;FOLD SLIN P257 Vel=1 m/s CPDAT257 Tool[4]:Microflown3D Base[0];%{PE}
;FOLD Parameters ;%{h}
;Params IlfProvider=kukaroboter.basistech.inlineforms.movement.spline; Kuka.IsGlobalPoint=False; Kuka.PointName=P257; Kuka.BlendingEnabled=False; Kuka.MoveDataName=CPDAT257; Kuka.VelocityPath=1.000; Kuka.VelocityFieldEnabled=True; Kuka.ColDetectFieldEnabled=True; Kuka.CurrentCDSetIndex=0; Kuka.MovementParameterFieldEnabled=True; IlfCommand=SLIN
;ENDFOLD
SLIN XP257 WITH $VEL = SVEL_CP(2.0, , LCPDAT257),$TOOL = STOOL2(FP257),$BASE = SBASE(FP257.BASE_NO),$IPO_MODE = SIPO_MODE(FP257.IPO_FRAME),$LOAD = SLOAD(FP257.TOOL_NO),$ACC = SACC_CP(LCPDAT257),$ORI_TYPE = SORI_TYP(LCPDAT257),$APO = SAPO(LCPDAT257),$JERK = SJERK(LCPDAT257),$COLLMON_TOL_PRO[1] = USE_CM_PRO_VALUES(0)
;ENDFOLD

;FOLD SLIN P258 Vel=1 m/s CPDAT258 Tool[4]:Microflown3D Base[0];%{PE}
;FOLD Parameters ;%{h}
;Params IlfProvider=kukaroboter.basistech.inlineforms.movement.spline; Kuka.IsGlobalPoint=False; Kuka.PointName=P258; Kuka.BlendingEnabled=False; Kuka.MoveDataName=CPDAT258; Kuka.VelocityPath=1.000; Kuka.VelocityFieldEnabled=True; Kuka.ColDetectFieldEnabled=True; Kuka.CurrentCDSetIndex=0; Kuka.MovementParameterFieldEnabled=True; IlfCommand=SLIN
;ENDFOLD
SLIN XP258 WITH $VEL = SVEL_CP(2.0, , LCPDAT258),$TOOL = STOOL2(FP258),$BASE = SBASE(FP258.BASE_NO),$IPO_MODE = SIPO_MODE(FP258.IPO_FRAME),$LOAD = SLOAD(FP258.TOOL_NO),$ACC = SACC_CP(LCPDAT258),$ORI_TYPE = SORI_TYP(LCPDAT258),$APO = SAPO(LCPDAT258),$JERK = SJERK(LCPDAT258),$COLLMON_TOL_PRO[1] = USE_CM_PRO_VALUES(0)
;ENDFOLD

;FOLD SLIN P259 Vel=1 m/s CPDAT259 Tool[4]:Microflown3D Base[0];%{PE}
;FOLD Parameters ;%{h}
;Params IlfProvider=kukaroboter.basistech.inlineforms.movement.spline; Kuka.IsGlobalPoint=False; Kuka.PointName=P259; Kuka.BlendingEnabled=False; Kuka.MoveDataName=CPDAT259; Kuka.VelocityPath=1.000; Kuka.VelocityFieldEnabled=True; Kuka.ColDetectFieldEnabled=True; Kuka.CurrentCDSetIndex=0; Kuka.MovementParameterFieldEnabled=True; IlfCommand=SLIN
;ENDFOLD
SLIN XP259 WITH $VEL = SVEL_CP(2.0, , LCPDAT259),$TOOL = STOOL2(FP259),$BASE = SBASE(FP259.BASE_NO),$IPO_MODE = SIPO_MODE(FP259.IPO_FRAME),$LOAD = SLOAD(FP259.TOOL_NO),$ACC = SACC_CP(LCPDAT259),$ORI_TYPE = SORI_TYP(LCPDAT259),$APO = SAPO(LCPDAT259),$JERK = SJERK(LCPDAT259),$COLLMON_TOL_PRO[1] = USE_CM_PRO_VALUES(0)
;ENDFOLD

;FOLD SLIN P260 Vel=1 m/s CPDAT260 Tool[4]:Microflown3D Base[0];%{PE}
;FOLD Parameters ;%{h}
;Params IlfProvider=kukaroboter.basistech.inlineforms.movement.spline; Kuka.IsGlobalPoint=False; Kuka.PointName=P260; Kuka.BlendingEnabled=False; Kuka.MoveDataName=CPDAT260; Kuka.VelocityPath=1.000; Kuka.VelocityFieldEnabled=True; Kuka.ColDetectFieldEnabled=True; Kuka.CurrentCDSetIndex=0; Kuka.MovementParameterFieldEnabled=True; IlfCommand=SLIN
;ENDFOLD
SLIN XP260 WITH $VEL = SVEL_CP(2.0, , LCPDAT260),$TOOL = STOOL2(FP260),$BASE = SBASE(FP260.BASE_NO),$IPO_MODE = SIPO_MODE(FP260.IPO_FRAME),$LOAD = SLOAD(FP260.TOOL_NO),$ACC = SACC_CP(LCPDAT260),$ORI_TYPE = SORI_TYP(LCPDAT260),$APO = SAPO(LCPDAT260),$JERK = SJERK(LCPDAT260),$COLLMON_TOL_PRO[1] = USE_CM_PRO_VALUES(0)
;ENDFOLD

;FOLD SLIN P261 Vel=1 m/s CPDAT261 Tool[4]:Microflown3D Base[0];%{PE}
;FOLD Parameters ;%{h}
;Params IlfProvider=kukaroboter.basistech.inlineforms.movement.spline; Kuka.IsGlobalPoint=False; Kuka.PointName=P261; Kuka.BlendingEnabled=False; Kuka.MoveDataName=CPDAT261; Kuka.VelocityPath=1.000; Kuka.VelocityFieldEnabled=True; Kuka.ColDetectFieldEnabled=True; Kuka.CurrentCDSetIndex=0; Kuka.MovementParameterFieldEnabled=True; IlfCommand=SLIN
;ENDFOLD
SLIN XP261 WITH $VEL = SVEL_CP(2.0, , LCPDAT261),$TOOL = STOOL2(FP261),$BASE = SBASE(FP261.BASE_NO),$IPO_MODE = SIPO_MODE(FP261.IPO_FRAME),$LOAD = SLOAD(FP261.TOOL_NO),$ACC = SACC_CP(LCPDAT261),$ORI_TYPE = SORI_TYP(LCPDAT261),$APO = SAPO(LCPDAT261),$JERK = SJERK(LCPDAT261),$COLLMON_TOL_PRO[1] = USE_CM_PRO_VALUES(0)
;ENDFOLD

;FOLD SLIN P262 Vel=1 m/s CPDAT262 Tool[4]:Microflown3D Base[0];%{PE}
;FOLD Parameters ;%{h}
;Params IlfProvider=kukaroboter.basistech.inlineforms.movement.spline; Kuka.IsGlobalPoint=False; Kuka.PointName=P262; Kuka.BlendingEnabled=False; Kuka.MoveDataName=CPDAT262; Kuka.VelocityPath=1.000; Kuka.VelocityFieldEnabled=True; Kuka.ColDetectFieldEnabled=True; Kuka.CurrentCDSetIndex=0; Kuka.MovementParameterFieldEnabled=True; IlfCommand=SLIN
;ENDFOLD
SLIN XP262 WITH $VEL = SVEL_CP(2.0, , LCPDAT262),$TOOL = STOOL2(FP262),$BASE = SBASE(FP262.BASE_NO),$IPO_MODE = SIPO_MODE(FP262.IPO_FRAME),$LOAD = SLOAD(FP262.TOOL_NO),$ACC = SACC_CP(LCPDAT262),$ORI_TYPE = SORI_TYP(LCPDAT262),$APO = SAPO(LCPDAT262),$JERK = SJERK(LCPDAT262),$COLLMON_TOL_PRO[1] = USE_CM_PRO_VALUES(0)
;ENDFOLD

;FOLD SLIN P263 Vel=1 m/s CPDAT263 Tool[4]:Microflown3D Base[0];%{PE}
;FOLD Parameters ;%{h}
;Params IlfProvider=kukaroboter.basistech.inlineforms.movement.spline; Kuka.IsGlobalPoint=False; Kuka.PointName=P263; Kuka.BlendingEnabled=False; Kuka.MoveDataName=CPDAT263; Kuka.VelocityPath=1.000; Kuka.VelocityFieldEnabled=True; Kuka.ColDetectFieldEnabled=True; Kuka.CurrentCDSetIndex=0; Kuka.MovementParameterFieldEnabled=True; IlfCommand=SLIN
;ENDFOLD
SLIN XP263 WITH $VEL = SVEL_CP(2.0, , LCPDAT263),$TOOL = STOOL2(FP263),$BASE = SBASE(FP263.BASE_NO),$IPO_MODE = SIPO_MODE(FP263.IPO_FRAME),$LOAD = SLOAD(FP263.TOOL_NO),$ACC = SACC_CP(LCPDAT263),$ORI_TYPE = SORI_TYP(LCPDAT263),$APO = SAPO(LCPDAT263),$JERK = SJERK(LCPDAT263),$COLLMON_TOL_PRO[1] = USE_CM_PRO_VALUES(0)
;ENDFOLD

;FOLD SLIN P264 Vel=1 m/s CPDAT264 Tool[4]:Microflown3D Base[0];%{PE}
;FOLD Parameters ;%{h}
;Params IlfProvider=kukaroboter.basistech.inlineforms.movement.spline; Kuka.IsGlobalPoint=False; Kuka.PointName=P264; Kuka.BlendingEnabled=False; Kuka.MoveDataName=CPDAT264; Kuka.VelocityPath=1.000; Kuka.VelocityFieldEnabled=True; Kuka.ColDetectFieldEnabled=True; Kuka.CurrentCDSetIndex=0; Kuka.MovementParameterFieldEnabled=True; IlfCommand=SLIN
;ENDFOLD
SLIN XP264 WITH $VEL = SVEL_CP(2.0, , LCPDAT264),$TOOL = STOOL2(FP264),$BASE = SBASE(FP264.BASE_NO),$IPO_MODE = SIPO_MODE(FP264.IPO_FRAME),$LOAD = SLOAD(FP264.TOOL_NO),$ACC = SACC_CP(LCPDAT264),$ORI_TYPE = SORI_TYP(LCPDAT264),$APO = SAPO(LCPDAT264),$JERK = SJERK(LCPDAT264),$COLLMON_TOL_PRO[1] = USE_CM_PRO_VALUES(0)
;ENDFOLD

;FOLD SLIN P265 Vel=1 m/s CPDAT265 Tool[4]:Microflown3D Base[0];%{PE}
;FOLD Parameters ;%{h}
;Params IlfProvider=kukaroboter.basistech.inlineforms.movement.spline; Kuka.IsGlobalPoint=False; Kuka.PointName=P265; Kuka.BlendingEnabled=False; Kuka.MoveDataName=CPDAT265; Kuka.VelocityPath=1.000; Kuka.VelocityFieldEnabled=True; Kuka.ColDetectFieldEnabled=True; Kuka.CurrentCDSetIndex=0; Kuka.MovementParameterFieldEnabled=True; IlfCommand=SLIN
;ENDFOLD
SLIN XP265 WITH $VEL = SVEL_CP(2.0, , LCPDAT265),$TOOL = STOOL2(FP265),$BASE = SBASE(FP265.BASE_NO),$IPO_MODE = SIPO_MODE(FP265.IPO_FRAME),$LOAD = SLOAD(FP265.TOOL_NO),$ACC = SACC_CP(LCPDAT265),$ORI_TYPE = SORI_TYP(LCPDAT265),$APO = SAPO(LCPDAT265),$JERK = SJERK(LCPDAT265),$COLLMON_TOL_PRO[1] = USE_CM_PRO_VALUES(0)
;ENDFOLD

;FOLD SLIN P266 Vel=1 m/s CPDAT266 Tool[4]:Microflown3D Base[0];%{PE}
;FOLD Parameters ;%{h}
;Params IlfProvider=kukaroboter.basistech.inlineforms.movement.spline; Kuka.IsGlobalPoint=False; Kuka.PointName=P266; Kuka.BlendingEnabled=False; Kuka.MoveDataName=CPDAT266; Kuka.VelocityPath=1.000; Kuka.VelocityFieldEnabled=True; Kuka.ColDetectFieldEnabled=True; Kuka.CurrentCDSetIndex=0; Kuka.MovementParameterFieldEnabled=True; IlfCommand=SLIN
;ENDFOLD
SLIN XP266 WITH $VEL = SVEL_CP(2.0, , LCPDAT266),$TOOL = STOOL2(FP266),$BASE = SBASE(FP266.BASE_NO),$IPO_MODE = SIPO_MODE(FP266.IPO_FRAME),$LOAD = SLOAD(FP266.TOOL_NO),$ACC = SACC_CP(LCPDAT266),$ORI_TYPE = SORI_TYP(LCPDAT266),$APO = SAPO(LCPDAT266),$JERK = SJERK(LCPDAT266),$COLLMON_TOL_PRO[1] = USE_CM_PRO_VALUES(0)
;ENDFOLD

;FOLD SLIN P267 Vel=1 m/s CPDAT267 Tool[4]:Microflown3D Base[0];%{PE}
;FOLD Parameters ;%{h}
;Params IlfProvider=kukaroboter.basistech.inlineforms.movement.spline; Kuka.IsGlobalPoint=False; Kuka.PointName=P267; Kuka.BlendingEnabled=False; Kuka.MoveDataName=CPDAT267; Kuka.VelocityPath=1.000; Kuka.VelocityFieldEnabled=True; Kuka.ColDetectFieldEnabled=True; Kuka.CurrentCDSetIndex=0; Kuka.MovementParameterFieldEnabled=True; IlfCommand=SLIN
;ENDFOLD
SLIN XP267 WITH $VEL = SVEL_CP(2.0, , LCPDAT267),$TOOL = STOOL2(FP267),$BASE = SBASE(FP267.BASE_NO),$IPO_MODE = SIPO_MODE(FP267.IPO_FRAME),$LOAD = SLOAD(FP267.TOOL_NO),$ACC = SACC_CP(LCPDAT267),$ORI_TYPE = SORI_TYP(LCPDAT267),$APO = SAPO(LCPDAT267),$JERK = SJERK(LCPDAT267),$COLLMON_TOL_PRO[1] = USE_CM_PRO_VALUES(0)
;ENDFOLD

;FOLD SLIN P268 Vel=1 m/s CPDAT268 Tool[4]:Microflown3D Base[0];%{PE}
;FOLD Parameters ;%{h}
;Params IlfProvider=kukaroboter.basistech.inlineforms.movement.spline; Kuka.IsGlobalPoint=False; Kuka.PointName=P268; Kuka.BlendingEnabled=False; Kuka.MoveDataName=CPDAT268; Kuka.VelocityPath=1.000; Kuka.VelocityFieldEnabled=True; Kuka.ColDetectFieldEnabled=True; Kuka.CurrentCDSetIndex=0; Kuka.MovementParameterFieldEnabled=True; IlfCommand=SLIN
;ENDFOLD
SLIN XP268 WITH $VEL = SVEL_CP(2.0, , LCPDAT268),$TOOL = STOOL2(FP268),$BASE = SBASE(FP268.BASE_NO),$IPO_MODE = SIPO_MODE(FP268.IPO_FRAME),$LOAD = SLOAD(FP268.TOOL_NO),$ACC = SACC_CP(LCPDAT268),$ORI_TYPE = SORI_TYP(LCPDAT268),$APO = SAPO(LCPDAT268),$JERK = SJERK(LCPDAT268),$COLLMON_TOL_PRO[1] = USE_CM_PRO_VALUES(0)
;ENDFOLD

;FOLD SLIN P269 Vel=1 m/s CPDAT269 Tool[4]:Microflown3D Base[0];%{PE}
;FOLD Parameters ;%{h}
;Params IlfProvider=kukaroboter.basistech.inlineforms.movement.spline; Kuka.IsGlobalPoint=False; Kuka.PointName=P269; Kuka.BlendingEnabled=False; Kuka.MoveDataName=CPDAT269; Kuka.VelocityPath=1.000; Kuka.VelocityFieldEnabled=True; Kuka.ColDetectFieldEnabled=True; Kuka.CurrentCDSetIndex=0; Kuka.MovementParameterFieldEnabled=True; IlfCommand=SLIN
;ENDFOLD
SLIN XP269 WITH $VEL = SVEL_CP(2.0, , LCPDAT269),$TOOL = STOOL2(FP269),$BASE = SBASE(FP269.BASE_NO),$IPO_MODE = SIPO_MODE(FP269.IPO_FRAME),$LOAD = SLOAD(FP269.TOOL_NO),$ACC = SACC_CP(LCPDAT269),$ORI_TYPE = SORI_TYP(LCPDAT269),$APO = SAPO(LCPDAT269),$JERK = SJERK(LCPDAT269),$COLLMON_TOL_PRO[1] = USE_CM_PRO_VALUES(0)
;ENDFOLD

;FOLD SLIN P270 Vel=1 m/s CPDAT270 Tool[4]:Microflown3D Base[0];%{PE}
;FOLD Parameters ;%{h}
;Params IlfProvider=kukaroboter.basistech.inlineforms.movement.spline; Kuka.IsGlobalPoint=False; Kuka.PointName=P270; Kuka.BlendingEnabled=False; Kuka.MoveDataName=CPDAT270; Kuka.VelocityPath=1.000; Kuka.VelocityFieldEnabled=True; Kuka.ColDetectFieldEnabled=True; Kuka.CurrentCDSetIndex=0; Kuka.MovementParameterFieldEnabled=True; IlfCommand=SLIN
;ENDFOLD
SLIN XP270 WITH $VEL = SVEL_CP(2.0, , LCPDAT270),$TOOL = STOOL2(FP270),$BASE = SBASE(FP270.BASE_NO),$IPO_MODE = SIPO_MODE(FP270.IPO_FRAME),$LOAD = SLOAD(FP270.TOOL_NO),$ACC = SACC_CP(LCPDAT270),$ORI_TYPE = SORI_TYP(LCPDAT270),$APO = SAPO(LCPDAT270),$JERK = SJERK(LCPDAT270),$COLLMON_TOL_PRO[1] = USE_CM_PRO_VALUES(0)
;ENDFOLD

;FOLD SLIN P271 Vel=1 m/s CPDAT271 Tool[4]:Microflown3D Base[0];%{PE}
;FOLD Parameters ;%{h}
;Params IlfProvider=kukaroboter.basistech.inlineforms.movement.spline; Kuka.IsGlobalPoint=False; Kuka.PointName=P271; Kuka.BlendingEnabled=False; Kuka.MoveDataName=CPDAT271; Kuka.VelocityPath=1.000; Kuka.VelocityFieldEnabled=True; Kuka.ColDetectFieldEnabled=True; Kuka.CurrentCDSetIndex=0; Kuka.MovementParameterFieldEnabled=True; IlfCommand=SLIN
;ENDFOLD
SLIN XP271 WITH $VEL = SVEL_CP(2.0, , LCPDAT271),$TOOL = STOOL2(FP271),$BASE = SBASE(FP271.BASE_NO),$IPO_MODE = SIPO_MODE(FP271.IPO_FRAME),$LOAD = SLOAD(FP271.TOOL_NO),$ACC = SACC_CP(LCPDAT271),$ORI_TYPE = SORI_TYP(LCPDAT271),$APO = SAPO(LCPDAT271),$JERK = SJERK(LCPDAT271),$COLLMON_TOL_PRO[1] = USE_CM_PRO_VALUES(0)
;ENDFOLD

;FOLD SLIN P272 Vel=1 m/s CPDAT272 Tool[4]:Microflown3D Base[0];%{PE}
;FOLD Parameters ;%{h}
;Params IlfProvider=kukaroboter.basistech.inlineforms.movement.spline; Kuka.IsGlobalPoint=False; Kuka.PointName=P272; Kuka.BlendingEnabled=False; Kuka.MoveDataName=CPDAT272; Kuka.VelocityPath=1.000; Kuka.VelocityFieldEnabled=True; Kuka.ColDetectFieldEnabled=True; Kuka.CurrentCDSetIndex=0; Kuka.MovementParameterFieldEnabled=True; IlfCommand=SLIN
;ENDFOLD
SLIN XP272 WITH $VEL = SVEL_CP(2.0, , LCPDAT272),$TOOL = STOOL2(FP272),$BASE = SBASE(FP272.BASE_NO),$IPO_MODE = SIPO_MODE(FP272.IPO_FRAME),$LOAD = SLOAD(FP272.TOOL_NO),$ACC = SACC_CP(LCPDAT272),$ORI_TYPE = SORI_TYP(LCPDAT272),$APO = SAPO(LCPDAT272),$JERK = SJERK(LCPDAT272),$COLLMON_TOL_PRO[1] = USE_CM_PRO_VALUES(0)
;ENDFOLD

;FOLD SLIN P273 Vel=1 m/s CPDAT273 Tool[4]:Microflown3D Base[0];%{PE}
;FOLD Parameters ;%{h}
;Params IlfProvider=kukaroboter.basistech.inlineforms.movement.spline; Kuka.IsGlobalPoint=False; Kuka.PointName=P273; Kuka.BlendingEnabled=False; Kuka.MoveDataName=CPDAT273; Kuka.VelocityPath=1.000; Kuka.VelocityFieldEnabled=True; Kuka.ColDetectFieldEnabled=True; Kuka.CurrentCDSetIndex=0; Kuka.MovementParameterFieldEnabled=True; IlfCommand=SLIN
;ENDFOLD
SLIN XP273 WITH $VEL = SVEL_CP(2.0, , LCPDAT273),$TOOL = STOOL2(FP273),$BASE = SBASE(FP273.BASE_NO),$IPO_MODE = SIPO_MODE(FP273.IPO_FRAME),$LOAD = SLOAD(FP273.TOOL_NO),$ACC = SACC_CP(LCPDAT273),$ORI_TYPE = SORI_TYP(LCPDAT273),$APO = SAPO(LCPDAT273),$JERK = SJERK(LCPDAT273),$COLLMON_TOL_PRO[1] = USE_CM_PRO_VALUES(0)
;ENDFOLD

;FOLD SLIN P274 Vel=1 m/s CPDAT274 Tool[4]:Microflown3D Base[0];%{PE}
;FOLD Parameters ;%{h}
;Params IlfProvider=kukaroboter.basistech.inlineforms.movement.spline; Kuka.IsGlobalPoint=False; Kuka.PointName=P274; Kuka.BlendingEnabled=False; Kuka.MoveDataName=CPDAT274; Kuka.VelocityPath=1.000; Kuka.VelocityFieldEnabled=True; Kuka.ColDetectFieldEnabled=True; Kuka.CurrentCDSetIndex=0; Kuka.MovementParameterFieldEnabled=True; IlfCommand=SLIN
;ENDFOLD
SLIN XP274 WITH $VEL = SVEL_CP(2.0, , LCPDAT274),$TOOL = STOOL2(FP274),$BASE = SBASE(FP274.BASE_NO),$IPO_MODE = SIPO_MODE(FP274.IPO_FRAME),$LOAD = SLOAD(FP274.TOOL_NO),$ACC = SACC_CP(LCPDAT274),$ORI_TYPE = SORI_TYP(LCPDAT274),$APO = SAPO(LCPDAT274),$JERK = SJERK(LCPDAT274),$COLLMON_TOL_PRO[1] = USE_CM_PRO_VALUES(0)
;ENDFOLD

;FOLD SLIN P275 Vel=1 m/s CPDAT275 Tool[4]:Microflown3D Base[0];%{PE}
;FOLD Parameters ;%{h}
;Params IlfProvider=kukaroboter.basistech.inlineforms.movement.spline; Kuka.IsGlobalPoint=False; Kuka.PointName=P275; Kuka.BlendingEnabled=False; Kuka.MoveDataName=CPDAT275; Kuka.VelocityPath=1.000; Kuka.VelocityFieldEnabled=True; Kuka.ColDetectFieldEnabled=True; Kuka.CurrentCDSetIndex=0; Kuka.MovementParameterFieldEnabled=True; IlfCommand=SLIN
;ENDFOLD
SLIN XP275 WITH $VEL = SVEL_CP(2.0, , LCPDAT275),$TOOL = STOOL2(FP275),$BASE = SBASE(FP275.BASE_NO),$IPO_MODE = SIPO_MODE(FP275.IPO_FRAME),$LOAD = SLOAD(FP275.TOOL_NO),$ACC = SACC_CP(LCPDAT275),$ORI_TYPE = SORI_TYP(LCPDAT275),$APO = SAPO(LCPDAT275),$JERK = SJERK(LCPDAT275),$COLLMON_TOL_PRO[1] = USE_CM_PRO_VALUES(0)
;ENDFOLD

;FOLD SLIN P276 Vel=1 m/s CPDAT276 Tool[4]:Microflown3D Base[0];%{PE}
;FOLD Parameters ;%{h}
;Params IlfProvider=kukaroboter.basistech.inlineforms.movement.spline; Kuka.IsGlobalPoint=False; Kuka.PointName=P276; Kuka.BlendingEnabled=False; Kuka.MoveDataName=CPDAT276; Kuka.VelocityPath=1.000; Kuka.VelocityFieldEnabled=True; Kuka.ColDetectFieldEnabled=True; Kuka.CurrentCDSetIndex=0; Kuka.MovementParameterFieldEnabled=True; IlfCommand=SLIN
;ENDFOLD
SLIN XP276 WITH $VEL = SVEL_CP(2.0, , LCPDAT276),$TOOL = STOOL2(FP276),$BASE = SBASE(FP276.BASE_NO),$IPO_MODE = SIPO_MODE(FP276.IPO_FRAME),$LOAD = SLOAD(FP276.TOOL_NO),$ACC = SACC_CP(LCPDAT276),$ORI_TYPE = SORI_TYP(LCPDAT276),$APO = SAPO(LCPDAT276),$JERK = SJERK(LCPDAT276),$COLLMON_TOL_PRO[1] = USE_CM_PRO_VALUES(0)
;ENDFOLD

;FOLD SLIN P277 Vel=1 m/s CPDAT277 Tool[4]:Microflown3D Base[0];%{PE}
;FOLD Parameters ;%{h}
;Params IlfProvider=kukaroboter.basistech.inlineforms.movement.spline; Kuka.IsGlobalPoint=False; Kuka.PointName=P277; Kuka.BlendingEnabled=False; Kuka.MoveDataName=CPDAT277; Kuka.VelocityPath=1.000; Kuka.VelocityFieldEnabled=True; Kuka.ColDetectFieldEnabled=True; Kuka.CurrentCDSetIndex=0; Kuka.MovementParameterFieldEnabled=True; IlfCommand=SLIN
;ENDFOLD
SLIN XP277 WITH $VEL = SVEL_CP(2.0, , LCPDAT277),$TOOL = STOOL2(FP277),$BASE = SBASE(FP277.BASE_NO),$IPO_MODE = SIPO_MODE(FP277.IPO_FRAME),$LOAD = SLOAD(FP277.TOOL_NO),$ACC = SACC_CP(LCPDAT277),$ORI_TYPE = SORI_TYP(LCPDAT277),$APO = SAPO(LCPDAT277),$JERK = SJERK(LCPDAT277),$COLLMON_TOL_PRO[1] = USE_CM_PRO_VALUES(0)
;ENDFOLD

;FOLD SLIN P278 Vel=1 m/s CPDAT278 Tool[4]:Microflown3D Base[0];%{PE}
;FOLD Parameters ;%{h}
;Params IlfProvider=kukaroboter.basistech.inlineforms.movement.spline; Kuka.IsGlobalPoint=False; Kuka.PointName=P278; Kuka.BlendingEnabled=False; Kuka.MoveDataName=CPDAT278; Kuka.VelocityPath=1.000; Kuka.VelocityFieldEnabled=True; Kuka.ColDetectFieldEnabled=True; Kuka.CurrentCDSetIndex=0; Kuka.MovementParameterFieldEnabled=True; IlfCommand=SLIN
;ENDFOLD
SLIN XP278 WITH $VEL = SVEL_CP(2.0, , LCPDAT278),$TOOL = STOOL2(FP278),$BASE = SBASE(FP278.BASE_NO),$IPO_MODE = SIPO_MODE(FP278.IPO_FRAME),$LOAD = SLOAD(FP278.TOOL_NO),$ACC = SACC_CP(LCPDAT278),$ORI_TYPE = SORI_TYP(LCPDAT278),$APO = SAPO(LCPDAT278),$JERK = SJERK(LCPDAT278),$COLLMON_TOL_PRO[1] = USE_CM_PRO_VALUES(0)
;ENDFOLD

;FOLD SLIN P279 Vel=1 m/s CPDAT279 Tool[4]:Microflown3D Base[0];%{PE}
;FOLD Parameters ;%{h}
;Params IlfProvider=kukaroboter.basistech.inlineforms.movement.spline; Kuka.IsGlobalPoint=False; Kuka.PointName=P279; Kuka.BlendingEnabled=False; Kuka.MoveDataName=CPDAT279; Kuka.VelocityPath=1.000; Kuka.VelocityFieldEnabled=True; Kuka.ColDetectFieldEnabled=True; Kuka.CurrentCDSetIndex=0; Kuka.MovementParameterFieldEnabled=True; IlfCommand=SLIN
;ENDFOLD
SLIN XP279 WITH $VEL = SVEL_CP(2.0, , LCPDAT279),$TOOL = STOOL2(FP279),$BASE = SBASE(FP279.BASE_NO),$IPO_MODE = SIPO_MODE(FP279.IPO_FRAME),$LOAD = SLOAD(FP279.TOOL_NO),$ACC = SACC_CP(LCPDAT279),$ORI_TYPE = SORI_TYP(LCPDAT279),$APO = SAPO(LCPDAT279),$JERK = SJERK(LCPDAT279),$COLLMON_TOL_PRO[1] = USE_CM_PRO_VALUES(0)
;ENDFOLD

;FOLD SLIN P280 Vel=1 m/s CPDAT280 Tool[4]:Microflown3D Base[0];%{PE}
;FOLD Parameters ;%{h}
;Params IlfProvider=kukaroboter.basistech.inlineforms.movement.spline; Kuka.IsGlobalPoint=False; Kuka.PointName=P280; Kuka.BlendingEnabled=False; Kuka.MoveDataName=CPDAT280; Kuka.VelocityPath=1.000; Kuka.VelocityFieldEnabled=True; Kuka.ColDetectFieldEnabled=True; Kuka.CurrentCDSetIndex=0; Kuka.MovementParameterFieldEnabled=True; IlfCommand=SLIN
;ENDFOLD
SLIN XP280 WITH $VEL = SVEL_CP(2.0, , LCPDAT280),$TOOL = STOOL2(FP280),$BASE = SBASE(FP280.BASE_NO),$IPO_MODE = SIPO_MODE(FP280.IPO_FRAME),$LOAD = SLOAD(FP280.TOOL_NO),$ACC = SACC_CP(LCPDAT280),$ORI_TYPE = SORI_TYP(LCPDAT280),$APO = SAPO(LCPDAT280),$JERK = SJERK(LCPDAT280),$COLLMON_TOL_PRO[1] = USE_CM_PRO_VALUES(0)
;ENDFOLD

;FOLD SLIN P281 Vel=1 m/s CPDAT281 Tool[4]:Microflown3D Base[0];%{PE}
;FOLD Parameters ;%{h}
;Params IlfProvider=kukaroboter.basistech.inlineforms.movement.spline; Kuka.IsGlobalPoint=False; Kuka.PointName=P281; Kuka.BlendingEnabled=False; Kuka.MoveDataName=CPDAT281; Kuka.VelocityPath=1.000; Kuka.VelocityFieldEnabled=True; Kuka.ColDetectFieldEnabled=True; Kuka.CurrentCDSetIndex=0; Kuka.MovementParameterFieldEnabled=True; IlfCommand=SLIN
;ENDFOLD
SLIN XP281 WITH $VEL = SVEL_CP(2.0, , LCPDAT281),$TOOL = STOOL2(FP281),$BASE = SBASE(FP281.BASE_NO),$IPO_MODE = SIPO_MODE(FP281.IPO_FRAME),$LOAD = SLOAD(FP281.TOOL_NO),$ACC = SACC_CP(LCPDAT281),$ORI_TYPE = SORI_TYP(LCPDAT281),$APO = SAPO(LCPDAT281),$JERK = SJERK(LCPDAT281),$COLLMON_TOL_PRO[1] = USE_CM_PRO_VALUES(0)
;ENDFOLD

;FOLD SLIN P282 Vel=1 m/s CPDAT282 Tool[4]:Microflown3D Base[0];%{PE}
;FOLD Parameters ;%{h}
;Params IlfProvider=kukaroboter.basistech.inlineforms.movement.spline; Kuka.IsGlobalPoint=False; Kuka.PointName=P282; Kuka.BlendingEnabled=False; Kuka.MoveDataName=CPDAT282; Kuka.VelocityPath=1.000; Kuka.VelocityFieldEnabled=True; Kuka.ColDetectFieldEnabled=True; Kuka.CurrentCDSetIndex=0; Kuka.MovementParameterFieldEnabled=True; IlfCommand=SLIN
;ENDFOLD
SLIN XP282 WITH $VEL = SVEL_CP(2.0, , LCPDAT282),$TOOL = STOOL2(FP282),$BASE = SBASE(FP282.BASE_NO),$IPO_MODE = SIPO_MODE(FP282.IPO_FRAME),$LOAD = SLOAD(FP282.TOOL_NO),$ACC = SACC_CP(LCPDAT282),$ORI_TYPE = SORI_TYP(LCPDAT282),$APO = SAPO(LCPDAT282),$JERK = SJERK(LCPDAT282),$COLLMON_TOL_PRO[1] = USE_CM_PRO_VALUES(0)
;ENDFOLD

;FOLD SLIN P283 Vel=1 m/s CPDAT283 Tool[4]:Microflown3D Base[0];%{PE}
;FOLD Parameters ;%{h}
;Params IlfProvider=kukaroboter.basistech.inlineforms.movement.spline; Kuka.IsGlobalPoint=False; Kuka.PointName=P283; Kuka.BlendingEnabled=False; Kuka.MoveDataName=CPDAT283; Kuka.VelocityPath=1.000; Kuka.VelocityFieldEnabled=True; Kuka.ColDetectFieldEnabled=True; Kuka.CurrentCDSetIndex=0; Kuka.MovementParameterFieldEnabled=True; IlfCommand=SLIN
;ENDFOLD
SLIN XP283 WITH $VEL = SVEL_CP(2.0, , LCPDAT283),$TOOL = STOOL2(FP283),$BASE = SBASE(FP283.BASE_NO),$IPO_MODE = SIPO_MODE(FP283.IPO_FRAME),$LOAD = SLOAD(FP283.TOOL_NO),$ACC = SACC_CP(LCPDAT283),$ORI_TYPE = SORI_TYP(LCPDAT283),$APO = SAPO(LCPDAT283),$JERK = SJERK(LCPDAT283),$COLLMON_TOL_PRO[1] = USE_CM_PRO_VALUES(0)
;ENDFOLD

;FOLD SLIN P284 Vel=1 m/s CPDAT284 Tool[4]:Microflown3D Base[0];%{PE}
;FOLD Parameters ;%{h}
;Params IlfProvider=kukaroboter.basistech.inlineforms.movement.spline; Kuka.IsGlobalPoint=False; Kuka.PointName=P284; Kuka.BlendingEnabled=False; Kuka.MoveDataName=CPDAT284; Kuka.VelocityPath=1.000; Kuka.VelocityFieldEnabled=True; Kuka.ColDetectFieldEnabled=True; Kuka.CurrentCDSetIndex=0; Kuka.MovementParameterFieldEnabled=True; IlfCommand=SLIN
;ENDFOLD
SLIN XP284 WITH $VEL = SVEL_CP(2.0, , LCPDAT284),$TOOL = STOOL2(FP284),$BASE = SBASE(FP284.BASE_NO),$IPO_MODE = SIPO_MODE(FP284.IPO_FRAME),$LOAD = SLOAD(FP284.TOOL_NO),$ACC = SACC_CP(LCPDAT284),$ORI_TYPE = SORI_TYP(LCPDAT284),$APO = SAPO(LCPDAT284),$JERK = SJERK(LCPDAT284),$COLLMON_TOL_PRO[1] = USE_CM_PRO_VALUES(0)
;ENDFOLD

;FOLD SLIN P285 Vel=1 m/s CPDAT285 Tool[4]:Microflown3D Base[0];%{PE}
;FOLD Parameters ;%{h}
;Params IlfProvider=kukaroboter.basistech.inlineforms.movement.spline; Kuka.IsGlobalPoint=False; Kuka.PointName=P285; Kuka.BlendingEnabled=False; Kuka.MoveDataName=CPDAT285; Kuka.VelocityPath=1.000; Kuka.VelocityFieldEnabled=True; Kuka.ColDetectFieldEnabled=True; Kuka.CurrentCDSetIndex=0; Kuka.MovementParameterFieldEnabled=True; IlfCommand=SLIN
;ENDFOLD
SLIN XP285 WITH $VEL = SVEL_CP(2.0, , LCPDAT285),$TOOL = STOOL2(FP285),$BASE = SBASE(FP285.BASE_NO),$IPO_MODE = SIPO_MODE(FP285.IPO_FRAME),$LOAD = SLOAD(FP285.TOOL_NO),$ACC = SACC_CP(LCPDAT285),$ORI_TYPE = SORI_TYP(LCPDAT285),$APO = SAPO(LCPDAT285),$JERK = SJERK(LCPDAT285),$COLLMON_TOL_PRO[1] = USE_CM_PRO_VALUES(0)
;ENDFOLD

;FOLD SLIN P286 Vel=1 m/s CPDAT286 Tool[4]:Microflown3D Base[0];%{PE}
;FOLD Parameters ;%{h}
;Params IlfProvider=kukaroboter.basistech.inlineforms.movement.spline; Kuka.IsGlobalPoint=False; Kuka.PointName=P286; Kuka.BlendingEnabled=False; Kuka.MoveDataName=CPDAT286; Kuka.VelocityPath=1.000; Kuka.VelocityFieldEnabled=True; Kuka.ColDetectFieldEnabled=True; Kuka.CurrentCDSetIndex=0; Kuka.MovementParameterFieldEnabled=True; IlfCommand=SLIN
;ENDFOLD
SLIN XP286 WITH $VEL = SVEL_CP(2.0, , LCPDAT286),$TOOL = STOOL2(FP286),$BASE = SBASE(FP286.BASE_NO),$IPO_MODE = SIPO_MODE(FP286.IPO_FRAME),$LOAD = SLOAD(FP286.TOOL_NO),$ACC = SACC_CP(LCPDAT286),$ORI_TYPE = SORI_TYP(LCPDAT286),$APO = SAPO(LCPDAT286),$JERK = SJERK(LCPDAT286),$COLLMON_TOL_PRO[1] = USE_CM_PRO_VALUES(0)
;ENDFOLD

;FOLD SLIN P287 Vel=1 m/s CPDAT287 Tool[4]:Microflown3D Base[0];%{PE}
;FOLD Parameters ;%{h}
;Params IlfProvider=kukaroboter.basistech.inlineforms.movement.spline; Kuka.IsGlobalPoint=False; Kuka.PointName=P287; Kuka.BlendingEnabled=False; Kuka.MoveDataName=CPDAT287; Kuka.VelocityPath=1.000; Kuka.VelocityFieldEnabled=True; Kuka.ColDetectFieldEnabled=True; Kuka.CurrentCDSetIndex=0; Kuka.MovementParameterFieldEnabled=True; IlfCommand=SLIN
;ENDFOLD
SLIN XP287 WITH $VEL = SVEL_CP(2.0, , LCPDAT287),$TOOL = STOOL2(FP287),$BASE = SBASE(FP287.BASE_NO),$IPO_MODE = SIPO_MODE(FP287.IPO_FRAME),$LOAD = SLOAD(FP287.TOOL_NO),$ACC = SACC_CP(LCPDAT287),$ORI_TYPE = SORI_TYP(LCPDAT287),$APO = SAPO(LCPDAT287),$JERK = SJERK(LCPDAT287),$COLLMON_TOL_PRO[1] = USE_CM_PRO_VALUES(0)
;ENDFOLD

;FOLD SLIN P288 Vel=1 m/s CPDAT288 Tool[4]:Microflown3D Base[0];%{PE}
;FOLD Parameters ;%{h}
;Params IlfProvider=kukaroboter.basistech.inlineforms.movement.spline; Kuka.IsGlobalPoint=False; Kuka.PointName=P288; Kuka.BlendingEnabled=False; Kuka.MoveDataName=CPDAT288; Kuka.VelocityPath=1.000; Kuka.VelocityFieldEnabled=True; Kuka.ColDetectFieldEnabled=True; Kuka.CurrentCDSetIndex=0; Kuka.MovementParameterFieldEnabled=True; IlfCommand=SLIN
;ENDFOLD
SLIN XP288 WITH $VEL = SVEL_CP(2.0, , LCPDAT288),$TOOL = STOOL2(FP288),$BASE = SBASE(FP288.BASE_NO),$IPO_MODE = SIPO_MODE(FP288.IPO_FRAME),$LOAD = SLOAD(FP288.TOOL_NO),$ACC = SACC_CP(LCPDAT288),$ORI_TYPE = SORI_TYP(LCPDAT288),$APO = SAPO(LCPDAT288),$JERK = SJERK(LCPDAT288),$COLLMON_TOL_PRO[1] = USE_CM_PRO_VALUES(0)
;ENDFOLD

;FOLD SLIN P289 Vel=1 m/s CPDAT289 Tool[4]:Microflown3D Base[0];%{PE}
;FOLD Parameters ;%{h}
;Params IlfProvider=kukaroboter.basistech.inlineforms.movement.spline; Kuka.IsGlobalPoint=False; Kuka.PointName=P289; Kuka.BlendingEnabled=False; Kuka.MoveDataName=CPDAT289; Kuka.VelocityPath=1.000; Kuka.VelocityFieldEnabled=True; Kuka.ColDetectFieldEnabled=True; Kuka.CurrentCDSetIndex=0; Kuka.MovementParameterFieldEnabled=True; IlfCommand=SLIN
;ENDFOLD
SLIN XP289 WITH $VEL = SVEL_CP(2.0, , LCPDAT289),$TOOL = STOOL2(FP289),$BASE = SBASE(FP289.BASE_NO),$IPO_MODE = SIPO_MODE(FP289.IPO_FRAME),$LOAD = SLOAD(FP289.TOOL_NO),$ACC = SACC_CP(LCPDAT289),$ORI_TYPE = SORI_TYP(LCPDAT289),$APO = SAPO(LCPDAT289),$JERK = SJERK(LCPDAT289),$COLLMON_TOL_PRO[1] = USE_CM_PRO_VALUES(0)
;ENDFOLD

;FOLD SLIN P290 Vel=1 m/s CPDAT290 Tool[4]:Microflown3D Base[0];%{PE}
;FOLD Parameters ;%{h}
;Params IlfProvider=kukaroboter.basistech.inlineforms.movement.spline; Kuka.IsGlobalPoint=False; Kuka.PointName=P290; Kuka.BlendingEnabled=False; Kuka.MoveDataName=CPDAT290; Kuka.VelocityPath=1.000; Kuka.VelocityFieldEnabled=True; Kuka.ColDetectFieldEnabled=True; Kuka.CurrentCDSetIndex=0; Kuka.MovementParameterFieldEnabled=True; IlfCommand=SLIN
;ENDFOLD
SLIN XP290 WITH $VEL = SVEL_CP(2.0, , LCPDAT290),$TOOL = STOOL2(FP290),$BASE = SBASE(FP290.BASE_NO),$IPO_MODE = SIPO_MODE(FP290.IPO_FRAME),$LOAD = SLOAD(FP290.TOOL_NO),$ACC = SACC_CP(LCPDAT290),$ORI_TYPE = SORI_TYP(LCPDAT290),$APO = SAPO(LCPDAT290),$JERK = SJERK(LCPDAT290),$COLLMON_TOL_PRO[1] = USE_CM_PRO_VALUES(0)
;ENDFOLD

;FOLD SLIN P291 Vel=1 m/s CPDAT291 Tool[4]:Microflown3D Base[0];%{PE}
;FOLD Parameters ;%{h}
;Params IlfProvider=kukaroboter.basistech.inlineforms.movement.spline; Kuka.IsGlobalPoint=False; Kuka.PointName=P291; Kuka.BlendingEnabled=False; Kuka.MoveDataName=CPDAT291; Kuka.VelocityPath=1.000; Kuka.VelocityFieldEnabled=True; Kuka.ColDetectFieldEnabled=True; Kuka.CurrentCDSetIndex=0; Kuka.MovementParameterFieldEnabled=True; IlfCommand=SLIN
;ENDFOLD
SLIN XP291 WITH $VEL = SVEL_CP(2.0, , LCPDAT291),$TOOL = STOOL2(FP291),$BASE = SBASE(FP291.BASE_NO),$IPO_MODE = SIPO_MODE(FP291.IPO_FRAME),$LOAD = SLOAD(FP291.TOOL_NO),$ACC = SACC_CP(LCPDAT291),$ORI_TYPE = SORI_TYP(LCPDAT291),$APO = SAPO(LCPDAT291),$JERK = SJERK(LCPDAT291),$COLLMON_TOL_PRO[1] = USE_CM_PRO_VALUES(0)
;ENDFOLD

;FOLD SLIN P292 Vel=1 m/s CPDAT292 Tool[4]:Microflown3D Base[0];%{PE}
;FOLD Parameters ;%{h}
;Params IlfProvider=kukaroboter.basistech.inlineforms.movement.spline; Kuka.IsGlobalPoint=False; Kuka.PointName=P292; Kuka.BlendingEnabled=False; Kuka.MoveDataName=CPDAT292; Kuka.VelocityPath=1.000; Kuka.VelocityFieldEnabled=True; Kuka.ColDetectFieldEnabled=True; Kuka.CurrentCDSetIndex=0; Kuka.MovementParameterFieldEnabled=True; IlfCommand=SLIN
;ENDFOLD
SLIN XP292 WITH $VEL = SVEL_CP(2.0, , LCPDAT292),$TOOL = STOOL2(FP292),$BASE = SBASE(FP292.BASE_NO),$IPO_MODE = SIPO_MODE(FP292.IPO_FRAME),$LOAD = SLOAD(FP292.TOOL_NO),$ACC = SACC_CP(LCPDAT292),$ORI_TYPE = SORI_TYP(LCPDAT292),$APO = SAPO(LCPDAT292),$JERK = SJERK(LCPDAT292),$COLLMON_TOL_PRO[1] = USE_CM_PRO_VALUES(0)
;ENDFOLD

;FOLD SLIN P293 Vel=1 m/s CPDAT293 Tool[4]:Microflown3D Base[0];%{PE}
;FOLD Parameters ;%{h}
;Params IlfProvider=kukaroboter.basistech.inlineforms.movement.spline; Kuka.IsGlobalPoint=False; Kuka.PointName=P293; Kuka.BlendingEnabled=False; Kuka.MoveDataName=CPDAT293; Kuka.VelocityPath=1.000; Kuka.VelocityFieldEnabled=True; Kuka.ColDetectFieldEnabled=True; Kuka.CurrentCDSetIndex=0; Kuka.MovementParameterFieldEnabled=True; IlfCommand=SLIN
;ENDFOLD
SLIN XP293 WITH $VEL = SVEL_CP(2.0, , LCPDAT293),$TOOL = STOOL2(FP293),$BASE = SBASE(FP293.BASE_NO),$IPO_MODE = SIPO_MODE(FP293.IPO_FRAME),$LOAD = SLOAD(FP293.TOOL_NO),$ACC = SACC_CP(LCPDAT293),$ORI_TYPE = SORI_TYP(LCPDAT293),$APO = SAPO(LCPDAT293),$JERK = SJERK(LCPDAT293),$COLLMON_TOL_PRO[1] = USE_CM_PRO_VALUES(0)
;ENDFOLD

;FOLD SLIN P294 Vel=1 m/s CPDAT294 Tool[4]:Microflown3D Base[0];%{PE}
;FOLD Parameters ;%{h}
;Params IlfProvider=kukaroboter.basistech.inlineforms.movement.spline; Kuka.IsGlobalPoint=False; Kuka.PointName=P294; Kuka.BlendingEnabled=False; Kuka.MoveDataName=CPDAT294; Kuka.VelocityPath=1.000; Kuka.VelocityFieldEnabled=True; Kuka.ColDetectFieldEnabled=True; Kuka.CurrentCDSetIndex=0; Kuka.MovementParameterFieldEnabled=True; IlfCommand=SLIN
;ENDFOLD
SLIN XP294 WITH $VEL = SVEL_CP(2.0, , LCPDAT294),$TOOL = STOOL2(FP294),$BASE = SBASE(FP294.BASE_NO),$IPO_MODE = SIPO_MODE(FP294.IPO_FRAME),$LOAD = SLOAD(FP294.TOOL_NO),$ACC = SACC_CP(LCPDAT294),$ORI_TYPE = SORI_TYP(LCPDAT294),$APO = SAPO(LCPDAT294),$JERK = SJERK(LCPDAT294),$COLLMON_TOL_PRO[1] = USE_CM_PRO_VALUES(0)
;ENDFOLD

;FOLD SLIN P295 Vel=1 m/s CPDAT295 Tool[4]:Microflown3D Base[0];%{PE}
;FOLD Parameters ;%{h}
;Params IlfProvider=kukaroboter.basistech.inlineforms.movement.spline; Kuka.IsGlobalPoint=False; Kuka.PointName=P295; Kuka.BlendingEnabled=False; Kuka.MoveDataName=CPDAT295; Kuka.VelocityPath=1.000; Kuka.VelocityFieldEnabled=True; Kuka.ColDetectFieldEnabled=True; Kuka.CurrentCDSetIndex=0; Kuka.MovementParameterFieldEnabled=True; IlfCommand=SLIN
;ENDFOLD
SLIN XP295 WITH $VEL = SVEL_CP(2.0, , LCPDAT295),$TOOL = STOOL2(FP295),$BASE = SBASE(FP295.BASE_NO),$IPO_MODE = SIPO_MODE(FP295.IPO_FRAME),$LOAD = SLOAD(FP295.TOOL_NO),$ACC = SACC_CP(LCPDAT295),$ORI_TYPE = SORI_TYP(LCPDAT295),$APO = SAPO(LCPDAT295),$JERK = SJERK(LCPDAT295),$COLLMON_TOL_PRO[1] = USE_CM_PRO_VALUES(0)
;ENDFOLD

;FOLD SLIN P296 Vel=1 m/s CPDAT296 Tool[4]:Microflown3D Base[0];%{PE}
;FOLD Parameters ;%{h}
;Params IlfProvider=kukaroboter.basistech.inlineforms.movement.spline; Kuka.IsGlobalPoint=False; Kuka.PointName=P296; Kuka.BlendingEnabled=False; Kuka.MoveDataName=CPDAT296; Kuka.VelocityPath=1.000; Kuka.VelocityFieldEnabled=True; Kuka.ColDetectFieldEnabled=True; Kuka.CurrentCDSetIndex=0; Kuka.MovementParameterFieldEnabled=True; IlfCommand=SLIN
;ENDFOLD
SLIN XP296 WITH $VEL = SVEL_CP(2.0, , LCPDAT296),$TOOL = STOOL2(FP296),$BASE = SBASE(FP296.BASE_NO),$IPO_MODE = SIPO_MODE(FP296.IPO_FRAME),$LOAD = SLOAD(FP296.TOOL_NO),$ACC = SACC_CP(LCPDAT296),$ORI_TYPE = SORI_TYP(LCPDAT296),$APO = SAPO(LCPDAT296),$JERK = SJERK(LCPDAT296),$COLLMON_TOL_PRO[1] = USE_CM_PRO_VALUES(0)
;ENDFOLD

;FOLD SLIN P297 Vel=1 m/s CPDAT297 Tool[4]:Microflown3D Base[0];%{PE}
;FOLD Parameters ;%{h}
;Params IlfProvider=kukaroboter.basistech.inlineforms.movement.spline; Kuka.IsGlobalPoint=False; Kuka.PointName=P297; Kuka.BlendingEnabled=False; Kuka.MoveDataName=CPDAT297; Kuka.VelocityPath=1.000; Kuka.VelocityFieldEnabled=True; Kuka.ColDetectFieldEnabled=True; Kuka.CurrentCDSetIndex=0; Kuka.MovementParameterFieldEnabled=True; IlfCommand=SLIN
;ENDFOLD
SLIN XP297 WITH $VEL = SVEL_CP(2.0, , LCPDAT297),$TOOL = STOOL2(FP297),$BASE = SBASE(FP297.BASE_NO),$IPO_MODE = SIPO_MODE(FP297.IPO_FRAME),$LOAD = SLOAD(FP297.TOOL_NO),$ACC = SACC_CP(LCPDAT297),$ORI_TYPE = SORI_TYP(LCPDAT297),$APO = SAPO(LCPDAT297),$JERK = SJERK(LCPDAT297),$COLLMON_TOL_PRO[1] = USE_CM_PRO_VALUES(0)
;ENDFOLD

;FOLD SLIN P298 Vel=1 m/s CPDAT298 Tool[4]:Microflown3D Base[0];%{PE}
;FOLD Parameters ;%{h}
;Params IlfProvider=kukaroboter.basistech.inlineforms.movement.spline; Kuka.IsGlobalPoint=False; Kuka.PointName=P298; Kuka.BlendingEnabled=False; Kuka.MoveDataName=CPDAT298; Kuka.VelocityPath=1.000; Kuka.VelocityFieldEnabled=True; Kuka.ColDetectFieldEnabled=True; Kuka.CurrentCDSetIndex=0; Kuka.MovementParameterFieldEnabled=True; IlfCommand=SLIN
;ENDFOLD
SLIN XP298 WITH $VEL = SVEL_CP(2.0, , LCPDAT298),$TOOL = STOOL2(FP298),$BASE = SBASE(FP298.BASE_NO),$IPO_MODE = SIPO_MODE(FP298.IPO_FRAME),$LOAD = SLOAD(FP298.TOOL_NO),$ACC = SACC_CP(LCPDAT298),$ORI_TYPE = SORI_TYP(LCPDAT298),$APO = SAPO(LCPDAT298),$JERK = SJERK(LCPDAT298),$COLLMON_TOL_PRO[1] = USE_CM_PRO_VALUES(0)
;ENDFOLD

;FOLD SLIN P299 Vel=1 m/s CPDAT299 Tool[4]:Microflown3D Base[0];%{PE}
;FOLD Parameters ;%{h}
;Params IlfProvider=kukaroboter.basistech.inlineforms.movement.spline; Kuka.IsGlobalPoint=False; Kuka.PointName=P299; Kuka.BlendingEnabled=False; Kuka.MoveDataName=CPDAT299; Kuka.VelocityPath=1.000; Kuka.VelocityFieldEnabled=True; Kuka.ColDetectFieldEnabled=True; Kuka.CurrentCDSetIndex=0; Kuka.MovementParameterFieldEnabled=True; IlfCommand=SLIN
;ENDFOLD
SLIN XP299 WITH $VEL = SVEL_CP(2.0, , LCPDAT299),$TOOL = STOOL2(FP299),$BASE = SBASE(FP299.BASE_NO),$IPO_MODE = SIPO_MODE(FP299.IPO_FRAME),$LOAD = SLOAD(FP299.TOOL_NO),$ACC = SACC_CP(LCPDAT299),$ORI_TYPE = SORI_TYP(LCPDAT299),$APO = SAPO(LCPDAT299),$JERK = SJERK(LCPDAT299),$COLLMON_TOL_PRO[1] = USE_CM_PRO_VALUES(0)
;ENDFOLD

;FOLD SLIN P300 Vel=1 m/s CPDAT300 Tool[4]:Microflown3D Base[0];%{PE}
;FOLD Parameters ;%{h}
;Params IlfProvider=kukaroboter.basistech.inlineforms.movement.spline; Kuka.IsGlobalPoint=False; Kuka.PointName=P300; Kuka.BlendingEnabled=False; Kuka.MoveDataName=CPDAT300; Kuka.VelocityPath=1.000; Kuka.VelocityFieldEnabled=True; Kuka.ColDetectFieldEnabled=True; Kuka.CurrentCDSetIndex=0; Kuka.MovementParameterFieldEnabled=True; IlfCommand=SLIN
;ENDFOLD
SLIN XP300 WITH $VEL = SVEL_CP(2.0, , LCPDAT300),$TOOL = STOOL2(FP300),$BASE = SBASE(FP300.BASE_NO),$IPO_MODE = SIPO_MODE(FP300.IPO_FRAME),$LOAD = SLOAD(FP300.TOOL_NO),$ACC = SACC_CP(LCPDAT300),$ORI_TYPE = SORI_TYP(LCPDAT300),$APO = SAPO(LCPDAT300),$JERK = SJERK(LCPDAT300),$COLLMON_TOL_PRO[1] = USE_CM_PRO_VALUES(0)
;ENDFOLD

;FOLD SLIN P301 Vel=1 m/s CPDAT301 Tool[4]:Microflown3D Base[0];%{PE}
;FOLD Parameters ;%{h}
;Params IlfProvider=kukaroboter.basistech.inlineforms.movement.spline; Kuka.IsGlobalPoint=False; Kuka.PointName=P301; Kuka.BlendingEnabled=False; Kuka.MoveDataName=CPDAT301; Kuka.VelocityPath=1.000; Kuka.VelocityFieldEnabled=True; Kuka.ColDetectFieldEnabled=True; Kuka.CurrentCDSetIndex=0; Kuka.MovementParameterFieldEnabled=True; IlfCommand=SLIN
;ENDFOLD
SLIN XP301 WITH $VEL = SVEL_CP(2.0, , LCPDAT301),$TOOL = STOOL2(FP301),$BASE = SBASE(FP301.BASE_NO),$IPO_MODE = SIPO_MODE(FP301.IPO_FRAME),$LOAD = SLOAD(FP301.TOOL_NO),$ACC = SACC_CP(LCPDAT301),$ORI_TYPE = SORI_TYP(LCPDAT301),$APO = SAPO(LCPDAT301),$JERK = SJERK(LCPDAT301),$COLLMON_TOL_PRO[1] = USE_CM_PRO_VALUES(0)
;ENDFOLD

;FOLD SLIN P302 Vel=1 m/s CPDAT302 Tool[4]:Microflown3D Base[0];%{PE}
;FOLD Parameters ;%{h}
;Params IlfProvider=kukaroboter.basistech.inlineforms.movement.spline; Kuka.IsGlobalPoint=False; Kuka.PointName=P302; Kuka.BlendingEnabled=False; Kuka.MoveDataName=CPDAT302; Kuka.VelocityPath=1.000; Kuka.VelocityFieldEnabled=True; Kuka.ColDetectFieldEnabled=True; Kuka.CurrentCDSetIndex=0; Kuka.MovementParameterFieldEnabled=True; IlfCommand=SLIN
;ENDFOLD
SLIN XP302 WITH $VEL = SVEL_CP(2.0, , LCPDAT302),$TOOL = STOOL2(FP302),$BASE = SBASE(FP302.BASE_NO),$IPO_MODE = SIPO_MODE(FP302.IPO_FRAME),$LOAD = SLOAD(FP302.TOOL_NO),$ACC = SACC_CP(LCPDAT302),$ORI_TYPE = SORI_TYP(LCPDAT302),$APO = SAPO(LCPDAT302),$JERK = SJERK(LCPDAT302),$COLLMON_TOL_PRO[1] = USE_CM_PRO_VALUES(0)
;ENDFOLD

;FOLD SLIN P303 Vel=1 m/s CPDAT303 Tool[4]:Microflown3D Base[0];%{PE}
;FOLD Parameters ;%{h}
;Params IlfProvider=kukaroboter.basistech.inlineforms.movement.spline; Kuka.IsGlobalPoint=False; Kuka.PointName=P303; Kuka.BlendingEnabled=False; Kuka.MoveDataName=CPDAT303; Kuka.VelocityPath=1.000; Kuka.VelocityFieldEnabled=True; Kuka.ColDetectFieldEnabled=True; Kuka.CurrentCDSetIndex=0; Kuka.MovementParameterFieldEnabled=True; IlfCommand=SLIN
;ENDFOLD
SLIN XP303 WITH $VEL = SVEL_CP(2.0, , LCPDAT303),$TOOL = STOOL2(FP303),$BASE = SBASE(FP303.BASE_NO),$IPO_MODE = SIPO_MODE(FP303.IPO_FRAME),$LOAD = SLOAD(FP303.TOOL_NO),$ACC = SACC_CP(LCPDAT303),$ORI_TYPE = SORI_TYP(LCPDAT303),$APO = SAPO(LCPDAT303),$JERK = SJERK(LCPDAT303),$COLLMON_TOL_PRO[1] = USE_CM_PRO_VALUES(0)
;ENDFOLD

;FOLD SLIN P304 Vel=1 m/s CPDAT304 Tool[4]:Microflown3D Base[0];%{PE}
;FOLD Parameters ;%{h}
;Params IlfProvider=kukaroboter.basistech.inlineforms.movement.spline; Kuka.IsGlobalPoint=False; Kuka.PointName=P304; Kuka.BlendingEnabled=False; Kuka.MoveDataName=CPDAT304; Kuka.VelocityPath=1.000; Kuka.VelocityFieldEnabled=True; Kuka.ColDetectFieldEnabled=True; Kuka.CurrentCDSetIndex=0; Kuka.MovementParameterFieldEnabled=True; IlfCommand=SLIN
;ENDFOLD
SLIN XP304 WITH $VEL = SVEL_CP(2.0, , LCPDAT304),$TOOL = STOOL2(FP304),$BASE = SBASE(FP304.BASE_NO),$IPO_MODE = SIPO_MODE(FP304.IPO_FRAME),$LOAD = SLOAD(FP304.TOOL_NO),$ACC = SACC_CP(LCPDAT304),$ORI_TYPE = SORI_TYP(LCPDAT304),$APO = SAPO(LCPDAT304),$JERK = SJERK(LCPDAT304),$COLLMON_TOL_PRO[1] = USE_CM_PRO_VALUES(0)
;ENDFOLD

;FOLD SLIN P305 Vel=1 m/s CPDAT305 Tool[4]:Microflown3D Base[0];%{PE}
;FOLD Parameters ;%{h}
;Params IlfProvider=kukaroboter.basistech.inlineforms.movement.spline; Kuka.IsGlobalPoint=False; Kuka.PointName=P305; Kuka.BlendingEnabled=False; Kuka.MoveDataName=CPDAT305; Kuka.VelocityPath=1.000; Kuka.VelocityFieldEnabled=True; Kuka.ColDetectFieldEnabled=True; Kuka.CurrentCDSetIndex=0; Kuka.MovementParameterFieldEnabled=True; IlfCommand=SLIN
;ENDFOLD
SLIN XP305 WITH $VEL = SVEL_CP(2.0, , LCPDAT305),$TOOL = STOOL2(FP305),$BASE = SBASE(FP305.BASE_NO),$IPO_MODE = SIPO_MODE(FP305.IPO_FRAME),$LOAD = SLOAD(FP305.TOOL_NO),$ACC = SACC_CP(LCPDAT305),$ORI_TYPE = SORI_TYP(LCPDAT305),$APO = SAPO(LCPDAT305),$JERK = SJERK(LCPDAT305),$COLLMON_TOL_PRO[1] = USE_CM_PRO_VALUES(0)
;ENDFOLD

;FOLD SLIN P306 Vel=1 m/s CPDAT306 Tool[4]:Microflown3D Base[0];%{PE}
;FOLD Parameters ;%{h}
;Params IlfProvider=kukaroboter.basistech.inlineforms.movement.spline; Kuka.IsGlobalPoint=False; Kuka.PointName=P306; Kuka.BlendingEnabled=False; Kuka.MoveDataName=CPDAT306; Kuka.VelocityPath=1.000; Kuka.VelocityFieldEnabled=True; Kuka.ColDetectFieldEnabled=True; Kuka.CurrentCDSetIndex=0; Kuka.MovementParameterFieldEnabled=True; IlfCommand=SLIN
;ENDFOLD
SLIN XP306 WITH $VEL = SVEL_CP(2.0, , LCPDAT306),$TOOL = STOOL2(FP306),$BASE = SBASE(FP306.BASE_NO),$IPO_MODE = SIPO_MODE(FP306.IPO_FRAME),$LOAD = SLOAD(FP306.TOOL_NO),$ACC = SACC_CP(LCPDAT306),$ORI_TYPE = SORI_TYP(LCPDAT306),$APO = SAPO(LCPDAT306),$JERK = SJERK(LCPDAT306),$COLLMON_TOL_PRO[1] = USE_CM_PRO_VALUES(0)
;ENDFOLD

;FOLD SLIN P307 Vel=1 m/s CPDAT307 Tool[4]:Microflown3D Base[0];%{PE}
;FOLD Parameters ;%{h}
;Params IlfProvider=kukaroboter.basistech.inlineforms.movement.spline; Kuka.IsGlobalPoint=False; Kuka.PointName=P307; Kuka.BlendingEnabled=False; Kuka.MoveDataName=CPDAT307; Kuka.VelocityPath=1.000; Kuka.VelocityFieldEnabled=True; Kuka.ColDetectFieldEnabled=True; Kuka.CurrentCDSetIndex=0; Kuka.MovementParameterFieldEnabled=True; IlfCommand=SLIN
;ENDFOLD
SLIN XP307 WITH $VEL = SVEL_CP(2.0, , LCPDAT307),$TOOL = STOOL2(FP307),$BASE = SBASE(FP307.BASE_NO),$IPO_MODE = SIPO_MODE(FP307.IPO_FRAME),$LOAD = SLOAD(FP307.TOOL_NO),$ACC = SACC_CP(LCPDAT307),$ORI_TYPE = SORI_TYP(LCPDAT307),$APO = SAPO(LCPDAT307),$JERK = SJERK(LCPDAT307),$COLLMON_TOL_PRO[1] = USE_CM_PRO_VALUES(0)
;ENDFOLD

;FOLD SLIN P308 Vel=1 m/s CPDAT308 Tool[4]:Microflown3D Base[0];%{PE}
;FOLD Parameters ;%{h}
;Params IlfProvider=kukaroboter.basistech.inlineforms.movement.spline; Kuka.IsGlobalPoint=False; Kuka.PointName=P308; Kuka.BlendingEnabled=False; Kuka.MoveDataName=CPDAT308; Kuka.VelocityPath=1.000; Kuka.VelocityFieldEnabled=True; Kuka.ColDetectFieldEnabled=True; Kuka.CurrentCDSetIndex=0; Kuka.MovementParameterFieldEnabled=True; IlfCommand=SLIN
;ENDFOLD
SLIN XP308 WITH $VEL = SVEL_CP(2.0, , LCPDAT308),$TOOL = STOOL2(FP308),$BASE = SBASE(FP308.BASE_NO),$IPO_MODE = SIPO_MODE(FP308.IPO_FRAME),$LOAD = SLOAD(FP308.TOOL_NO),$ACC = SACC_CP(LCPDAT308),$ORI_TYPE = SORI_TYP(LCPDAT308),$APO = SAPO(LCPDAT308),$JERK = SJERK(LCPDAT308),$COLLMON_TOL_PRO[1] = USE_CM_PRO_VALUES(0)
;ENDFOLD

;FOLD SLIN P309 Vel=1 m/s CPDAT309 Tool[4]:Microflown3D Base[0];%{PE}
;FOLD Parameters ;%{h}
;Params IlfProvider=kukaroboter.basistech.inlineforms.movement.spline; Kuka.IsGlobalPoint=False; Kuka.PointName=P309; Kuka.BlendingEnabled=False; Kuka.MoveDataName=CPDAT309; Kuka.VelocityPath=1.000; Kuka.VelocityFieldEnabled=True; Kuka.ColDetectFieldEnabled=True; Kuka.CurrentCDSetIndex=0; Kuka.MovementParameterFieldEnabled=True; IlfCommand=SLIN
;ENDFOLD
SLIN XP309 WITH $VEL = SVEL_CP(2.0, , LCPDAT309),$TOOL = STOOL2(FP309),$BASE = SBASE(FP309.BASE_NO),$IPO_MODE = SIPO_MODE(FP309.IPO_FRAME),$LOAD = SLOAD(FP309.TOOL_NO),$ACC = SACC_CP(LCPDAT309),$ORI_TYPE = SORI_TYP(LCPDAT309),$APO = SAPO(LCPDAT309),$JERK = SJERK(LCPDAT309),$COLLMON_TOL_PRO[1] = USE_CM_PRO_VALUES(0)
;ENDFOLD

;FOLD SLIN P310 Vel=1 m/s CPDAT310 Tool[4]:Microflown3D Base[0];%{PE}
;FOLD Parameters ;%{h}
;Params IlfProvider=kukaroboter.basistech.inlineforms.movement.spline; Kuka.IsGlobalPoint=False; Kuka.PointName=P310; Kuka.BlendingEnabled=False; Kuka.MoveDataName=CPDAT310; Kuka.VelocityPath=1.000; Kuka.VelocityFieldEnabled=True; Kuka.ColDetectFieldEnabled=True; Kuka.CurrentCDSetIndex=0; Kuka.MovementParameterFieldEnabled=True; IlfCommand=SLIN
;ENDFOLD
SLIN XP310 WITH $VEL = SVEL_CP(2.0, , LCPDAT310),$TOOL = STOOL2(FP310),$BASE = SBASE(FP310.BASE_NO),$IPO_MODE = SIPO_MODE(FP310.IPO_FRAME),$LOAD = SLOAD(FP310.TOOL_NO),$ACC = SACC_CP(LCPDAT310),$ORI_TYPE = SORI_TYP(LCPDAT310),$APO = SAPO(LCPDAT310),$JERK = SJERK(LCPDAT310),$COLLMON_TOL_PRO[1] = USE_CM_PRO_VALUES(0)
;ENDFOLD

;FOLD SLIN P311 Vel=1 m/s CPDAT311 Tool[4]:Microflown3D Base[0];%{PE}
;FOLD Parameters ;%{h}
;Params IlfProvider=kukaroboter.basistech.inlineforms.movement.spline; Kuka.IsGlobalPoint=False; Kuka.PointName=P311; Kuka.BlendingEnabled=False; Kuka.MoveDataName=CPDAT311; Kuka.VelocityPath=1.000; Kuka.VelocityFieldEnabled=True; Kuka.ColDetectFieldEnabled=True; Kuka.CurrentCDSetIndex=0; Kuka.MovementParameterFieldEnabled=True; IlfCommand=SLIN
;ENDFOLD
SLIN XP311 WITH $VEL = SVEL_CP(2.0, , LCPDAT311),$TOOL = STOOL2(FP311),$BASE = SBASE(FP311.BASE_NO),$IPO_MODE = SIPO_MODE(FP311.IPO_FRAME),$LOAD = SLOAD(FP311.TOOL_NO),$ACC = SACC_CP(LCPDAT311),$ORI_TYPE = SORI_TYP(LCPDAT311),$APO = SAPO(LCPDAT311),$JERK = SJERK(LCPDAT311),$COLLMON_TOL_PRO[1] = USE_CM_PRO_VALUES(0)
;ENDFOLD

;FOLD SLIN P312 Vel=1 m/s CPDAT312 Tool[4]:Microflown3D Base[0];%{PE}
;FOLD Parameters ;%{h}
;Params IlfProvider=kukaroboter.basistech.inlineforms.movement.spline; Kuka.IsGlobalPoint=False; Kuka.PointName=P312; Kuka.BlendingEnabled=False; Kuka.MoveDataName=CPDAT312; Kuka.VelocityPath=1.000; Kuka.VelocityFieldEnabled=True; Kuka.ColDetectFieldEnabled=True; Kuka.CurrentCDSetIndex=0; Kuka.MovementParameterFieldEnabled=True; IlfCommand=SLIN
;ENDFOLD
SLIN XP312 WITH $VEL = SVEL_CP(2.0, , LCPDAT312),$TOOL = STOOL2(FP312),$BASE = SBASE(FP312.BASE_NO),$IPO_MODE = SIPO_MODE(FP312.IPO_FRAME),$LOAD = SLOAD(FP312.TOOL_NO),$ACC = SACC_CP(LCPDAT312),$ORI_TYPE = SORI_TYP(LCPDAT312),$APO = SAPO(LCPDAT312),$JERK = SJERK(LCPDAT312),$COLLMON_TOL_PRO[1] = USE_CM_PRO_VALUES(0)
;ENDFOLD

;FOLD SLIN P313 Vel=1 m/s CPDAT313 Tool[4]:Microflown3D Base[0];%{PE}
;FOLD Parameters ;%{h}
;Params IlfProvider=kukaroboter.basistech.inlineforms.movement.spline; Kuka.IsGlobalPoint=False; Kuka.PointName=P313; Kuka.BlendingEnabled=False; Kuka.MoveDataName=CPDAT313; Kuka.VelocityPath=1.000; Kuka.VelocityFieldEnabled=True; Kuka.ColDetectFieldEnabled=True; Kuka.CurrentCDSetIndex=0; Kuka.MovementParameterFieldEnabled=True; IlfCommand=SLIN
;ENDFOLD
SLIN XP313 WITH $VEL = SVEL_CP(2.0, , LCPDAT313),$TOOL = STOOL2(FP313),$BASE = SBASE(FP313.BASE_NO),$IPO_MODE = SIPO_MODE(FP313.IPO_FRAME),$LOAD = SLOAD(FP313.TOOL_NO),$ACC = SACC_CP(LCPDAT313),$ORI_TYPE = SORI_TYP(LCPDAT313),$APO = SAPO(LCPDAT313),$JERK = SJERK(LCPDAT313),$COLLMON_TOL_PRO[1] = USE_CM_PRO_VALUES(0)
;ENDFOLD

;FOLD SLIN P314 Vel=1 m/s CPDAT314 Tool[4]:Microflown3D Base[0];%{PE}
;FOLD Parameters ;%{h}
;Params IlfProvider=kukaroboter.basistech.inlineforms.movement.spline; Kuka.IsGlobalPoint=False; Kuka.PointName=P314; Kuka.BlendingEnabled=False; Kuka.MoveDataName=CPDAT314; Kuka.VelocityPath=1.000; Kuka.VelocityFieldEnabled=True; Kuka.ColDetectFieldEnabled=True; Kuka.CurrentCDSetIndex=0; Kuka.MovementParameterFieldEnabled=True; IlfCommand=SLIN
;ENDFOLD
SLIN XP314 WITH $VEL = SVEL_CP(2.0, , LCPDAT314),$TOOL = STOOL2(FP314),$BASE = SBASE(FP314.BASE_NO),$IPO_MODE = SIPO_MODE(FP314.IPO_FRAME),$LOAD = SLOAD(FP314.TOOL_NO),$ACC = SACC_CP(LCPDAT314),$ORI_TYPE = SORI_TYP(LCPDAT314),$APO = SAPO(LCPDAT314),$JERK = SJERK(LCPDAT314),$COLLMON_TOL_PRO[1] = USE_CM_PRO_VALUES(0)
;ENDFOLD

;FOLD SLIN P315 Vel=1 m/s CPDAT315 Tool[4]:Microflown3D Base[0];%{PE}
;FOLD Parameters ;%{h}
;Params IlfProvider=kukaroboter.basistech.inlineforms.movement.spline; Kuka.IsGlobalPoint=False; Kuka.PointName=P315; Kuka.BlendingEnabled=False; Kuka.MoveDataName=CPDAT315; Kuka.VelocityPath=1.000; Kuka.VelocityFieldEnabled=True; Kuka.ColDetectFieldEnabled=True; Kuka.CurrentCDSetIndex=0; Kuka.MovementParameterFieldEnabled=True; IlfCommand=SLIN
;ENDFOLD
SLIN XP315 WITH $VEL = SVEL_CP(2.0, , LCPDAT315),$TOOL = STOOL2(FP315),$BASE = SBASE(FP315.BASE_NO),$IPO_MODE = SIPO_MODE(FP315.IPO_FRAME),$LOAD = SLOAD(FP315.TOOL_NO),$ACC = SACC_CP(LCPDAT315),$ORI_TYPE = SORI_TYP(LCPDAT315),$APO = SAPO(LCPDAT315),$JERK = SJERK(LCPDAT315),$COLLMON_TOL_PRO[1] = USE_CM_PRO_VALUES(0)
;ENDFOLD

;FOLD SLIN P316 Vel=0.25 m/s CPDAT316 Tool[4]:Microflown3D Base[0];%{PE}
;FOLD Parameters ;%{h}
;Params IlfProvider=kukaroboter.basistech.inlineforms.movement.spline; Kuka.IsGlobalPoint=False; Kuka.PointName=P316; Kuka.BlendingEnabled=False; Kuka.MoveDataName=CPDAT316; Kuka.VelocityPath=0.250; Kuka.VelocityFieldEnabled=True; Kuka.ColDetectFieldEnabled=True; Kuka.CurrentCDSetIndex=0; Kuka.MovementParameterFieldEnabled=True; IlfCommand=SLIN
;ENDFOLD
SLIN XP316 WITH $VEL = SVEL_CP(2.0, , LCPDAT316),$TOOL = STOOL2(FP316),$BASE = SBASE(FP316.BASE_NO),$IPO_MODE = SIPO_MODE(FP316.IPO_FRAME),$LOAD = SLOAD(FP316.TOOL_NO),$ACC = SACC_CP(LCPDAT316),$ORI_TYPE = SORI_TYP(LCPDAT316),$APO = SAPO(LCPDAT316),$JERK = SJERK(LCPDAT316),$COLLMON_TOL_PRO[1] = USE_CM_PRO_VALUES(0)
;ENDFOLD

;FOLD SPTP P317 Vel=20 % PDAT317 Tool[4]:Microflown3D Base[0];%{PE}
;FOLD Parameters ;%{h}
;ParamsIlfProvider=kukaroboter.basistech.inlineforms.movement.spline; Kuka.IsGlobalPoint=False; Kuka.PointName=P317; Kuka.BlendingEnabled=False; Kuka.MoveDataPtpName=PDAT317; Kuka.VelocityPtp=20; Kuka.VelocityFieldEnabled=True; Kuka.ColDetectFieldEnabled=True; Kuka.CurrentCDSetIndex=0; Kuka.MovementParameterFieldEnabled=True; IlfCommand=SPTP
;ENDFOLD
SPTP XP317 WITH $VEL_AXIS[1] = SVEL_JOINT(20.0), $TOOL = STOOL2(FP317), $BASE = SBASE(FP317.BASE_NO), $IPO_MODE = SIPO_MODE(FP317.IPO_FRAME), $LOAD = SLOAD(FP317.TOOL_NO), $ACC_AXIS[1] = SACC_JOINT(PPDAT317), $APO = SAPO_PTP(PPDAT317), $GEAR_JERK[1] = SGEAR_JERK(PPDAT317), $COLLMON_TOL_PRO[1] = USE_CM_PRO_VALUES(0)
;ENDFOLD

;FOLD SLIN P318 Vel=0.25 m/s CPDAT318 Tool[4]:Microflown3D Base[0];%{PE}
;FOLD Parameters ;%{h}
;Params IlfProvider=kukaroboter.basistech.inlineforms.movement.spline; Kuka.IsGlobalPoint=False; Kuka.PointName=P318; Kuka.BlendingEnabled=False; Kuka.MoveDataName=CPDAT318; Kuka.VelocityPath=0.250; Kuka.VelocityFieldEnabled=True; Kuka.ColDetectFieldEnabled=True; Kuka.CurrentCDSetIndex=0; Kuka.MovementParameterFieldEnabled=True; IlfCommand=SLIN
;ENDFOLD
SLIN XP318 WITH $VEL = SVEL_CP(2.0, , LCPDAT318),$TOOL = STOOL2(FP318),$BASE = SBASE(FP318.BASE_NO),$IPO_MODE = SIPO_MODE(FP318.IPO_FRAME),$LOAD = SLOAD(FP318.TOOL_NO),$ACC = SACC_CP(LCPDAT318),$ORI_TYPE = SORI_TYP(LCPDAT318),$APO = SAPO(LCPDAT318),$JERK = SJERK(LCPDAT318),$COLLMON_TOL_PRO[1] = USE_CM_PRO_VALUES(0)
;ENDFOLD

;FOLD SLIN P319 Vel=1 m/s CPDAT319 Tool[4]:Microflown3D Base[0];%{PE}
;FOLD Parameters ;%{h}
;Params IlfProvider=kukaroboter.basistech.inlineforms.movement.spline; Kuka.IsGlobalPoint=False; Kuka.PointName=P319; Kuka.BlendingEnabled=False; Kuka.MoveDataName=CPDAT319; Kuka.VelocityPath=1.000; Kuka.VelocityFieldEnabled=True; Kuka.ColDetectFieldEnabled=True; Kuka.CurrentCDSetIndex=0; Kuka.MovementParameterFieldEnabled=True; IlfCommand=SLIN
;ENDFOLD
SLIN XP319 WITH $VEL = SVEL_CP(2.0, , LCPDAT319),$TOOL = STOOL2(FP319),$BASE = SBASE(FP319.BASE_NO),$IPO_MODE = SIPO_MODE(FP319.IPO_FRAME),$LOAD = SLOAD(FP319.TOOL_NO),$ACC = SACC_CP(LCPDAT319),$ORI_TYPE = SORI_TYP(LCPDAT319),$APO = SAPO(LCPDAT319),$JERK = SJERK(LCPDAT319),$COLLMON_TOL_PRO[1] = USE_CM_PRO_VALUES(0)
;ENDFOLD

;FOLD SLIN P320 Vel=1 m/s CPDAT320 Tool[4]:Microflown3D Base[0];%{PE}
;FOLD Parameters ;%{h}
;Params IlfProvider=kukaroboter.basistech.inlineforms.movement.spline; Kuka.IsGlobalPoint=False; Kuka.PointName=P320; Kuka.BlendingEnabled=False; Kuka.MoveDataName=CPDAT320; Kuka.VelocityPath=1.000; Kuka.VelocityFieldEnabled=True; Kuka.ColDetectFieldEnabled=True; Kuka.CurrentCDSetIndex=0; Kuka.MovementParameterFieldEnabled=True; IlfCommand=SLIN
;ENDFOLD
SLIN XP320 WITH $VEL = SVEL_CP(2.0, , LCPDAT320),$TOOL = STOOL2(FP320),$BASE = SBASE(FP320.BASE_NO),$IPO_MODE = SIPO_MODE(FP320.IPO_FRAME),$LOAD = SLOAD(FP320.TOOL_NO),$ACC = SACC_CP(LCPDAT320),$ORI_TYPE = SORI_TYP(LCPDAT320),$APO = SAPO(LCPDAT320),$JERK = SJERK(LCPDAT320),$COLLMON_TOL_PRO[1] = USE_CM_PRO_VALUES(0)
;ENDFOLD

;FOLD SLIN P321 Vel=1 m/s CPDAT321 Tool[4]:Microflown3D Base[0];%{PE}
;FOLD Parameters ;%{h}
;Params IlfProvider=kukaroboter.basistech.inlineforms.movement.spline; Kuka.IsGlobalPoint=False; Kuka.PointName=P321; Kuka.BlendingEnabled=False; Kuka.MoveDataName=CPDAT321; Kuka.VelocityPath=1.000; Kuka.VelocityFieldEnabled=True; Kuka.ColDetectFieldEnabled=True; Kuka.CurrentCDSetIndex=0; Kuka.MovementParameterFieldEnabled=True; IlfCommand=SLIN
;ENDFOLD
SLIN XP321 WITH $VEL = SVEL_CP(2.0, , LCPDAT321),$TOOL = STOOL2(FP321),$BASE = SBASE(FP321.BASE_NO),$IPO_MODE = SIPO_MODE(FP321.IPO_FRAME),$LOAD = SLOAD(FP321.TOOL_NO),$ACC = SACC_CP(LCPDAT321),$ORI_TYPE = SORI_TYP(LCPDAT321),$APO = SAPO(LCPDAT321),$JERK = SJERK(LCPDAT321),$COLLMON_TOL_PRO[1] = USE_CM_PRO_VALUES(0)
;ENDFOLD

;FOLD SLIN P322 Vel=1 m/s CPDAT322 Tool[4]:Microflown3D Base[0];%{PE}
;FOLD Parameters ;%{h}
;Params IlfProvider=kukaroboter.basistech.inlineforms.movement.spline; Kuka.IsGlobalPoint=False; Kuka.PointName=P322; Kuka.BlendingEnabled=False; Kuka.MoveDataName=CPDAT322; Kuka.VelocityPath=1.000; Kuka.VelocityFieldEnabled=True; Kuka.ColDetectFieldEnabled=True; Kuka.CurrentCDSetIndex=0; Kuka.MovementParameterFieldEnabled=True; IlfCommand=SLIN
;ENDFOLD
SLIN XP322 WITH $VEL = SVEL_CP(2.0, , LCPDAT322),$TOOL = STOOL2(FP322),$BASE = SBASE(FP322.BASE_NO),$IPO_MODE = SIPO_MODE(FP322.IPO_FRAME),$LOAD = SLOAD(FP322.TOOL_NO),$ACC = SACC_CP(LCPDAT322),$ORI_TYPE = SORI_TYP(LCPDAT322),$APO = SAPO(LCPDAT322),$JERK = SJERK(LCPDAT322),$COLLMON_TOL_PRO[1] = USE_CM_PRO_VALUES(0)
;ENDFOLD

;FOLD SLIN P323 Vel=1 m/s CPDAT323 Tool[4]:Microflown3D Base[0];%{PE}
;FOLD Parameters ;%{h}
;Params IlfProvider=kukaroboter.basistech.inlineforms.movement.spline; Kuka.IsGlobalPoint=False; Kuka.PointName=P323; Kuka.BlendingEnabled=False; Kuka.MoveDataName=CPDAT323; Kuka.VelocityPath=1.000; Kuka.VelocityFieldEnabled=True; Kuka.ColDetectFieldEnabled=True; Kuka.CurrentCDSetIndex=0; Kuka.MovementParameterFieldEnabled=True; IlfCommand=SLIN
;ENDFOLD
SLIN XP323 WITH $VEL = SVEL_CP(2.0, , LCPDAT323),$TOOL = STOOL2(FP323),$BASE = SBASE(FP323.BASE_NO),$IPO_MODE = SIPO_MODE(FP323.IPO_FRAME),$LOAD = SLOAD(FP323.TOOL_NO),$ACC = SACC_CP(LCPDAT323),$ORI_TYPE = SORI_TYP(LCPDAT323),$APO = SAPO(LCPDAT323),$JERK = SJERK(LCPDAT323),$COLLMON_TOL_PRO[1] = USE_CM_PRO_VALUES(0)
;ENDFOLD

;FOLD SLIN P324 Vel=1 m/s CPDAT324 Tool[4]:Microflown3D Base[0];%{PE}
;FOLD Parameters ;%{h}
;Params IlfProvider=kukaroboter.basistech.inlineforms.movement.spline; Kuka.IsGlobalPoint=False; Kuka.PointName=P324; Kuka.BlendingEnabled=False; Kuka.MoveDataName=CPDAT324; Kuka.VelocityPath=1.000; Kuka.VelocityFieldEnabled=True; Kuka.ColDetectFieldEnabled=True; Kuka.CurrentCDSetIndex=0; Kuka.MovementParameterFieldEnabled=True; IlfCommand=SLIN
;ENDFOLD
SLIN XP324 WITH $VEL = SVEL_CP(2.0, , LCPDAT324),$TOOL = STOOL2(FP324),$BASE = SBASE(FP324.BASE_NO),$IPO_MODE = SIPO_MODE(FP324.IPO_FRAME),$LOAD = SLOAD(FP324.TOOL_NO),$ACC = SACC_CP(LCPDAT324),$ORI_TYPE = SORI_TYP(LCPDAT324),$APO = SAPO(LCPDAT324),$JERK = SJERK(LCPDAT324),$COLLMON_TOL_PRO[1] = USE_CM_PRO_VALUES(0)
;ENDFOLD

;FOLD SLIN P325 Vel=1 m/s CPDAT325 Tool[4]:Microflown3D Base[0];%{PE}
;FOLD Parameters ;%{h}
;Params IlfProvider=kukaroboter.basistech.inlineforms.movement.spline; Kuka.IsGlobalPoint=False; Kuka.PointName=P325; Kuka.BlendingEnabled=False; Kuka.MoveDataName=CPDAT325; Kuka.VelocityPath=1.000; Kuka.VelocityFieldEnabled=True; Kuka.ColDetectFieldEnabled=True; Kuka.CurrentCDSetIndex=0; Kuka.MovementParameterFieldEnabled=True; IlfCommand=SLIN
;ENDFOLD
SLIN XP325 WITH $VEL = SVEL_CP(2.0, , LCPDAT325),$TOOL = STOOL2(FP325),$BASE = SBASE(FP325.BASE_NO),$IPO_MODE = SIPO_MODE(FP325.IPO_FRAME),$LOAD = SLOAD(FP325.TOOL_NO),$ACC = SACC_CP(LCPDAT325),$ORI_TYPE = SORI_TYP(LCPDAT325),$APO = SAPO(LCPDAT325),$JERK = SJERK(LCPDAT325),$COLLMON_TOL_PRO[1] = USE_CM_PRO_VALUES(0)
;ENDFOLD

;FOLD SLIN P326 Vel=1 m/s CPDAT326 Tool[4]:Microflown3D Base[0];%{PE}
;FOLD Parameters ;%{h}
;Params IlfProvider=kukaroboter.basistech.inlineforms.movement.spline; Kuka.IsGlobalPoint=False; Kuka.PointName=P326; Kuka.BlendingEnabled=False; Kuka.MoveDataName=CPDAT326; Kuka.VelocityPath=1.000; Kuka.VelocityFieldEnabled=True; Kuka.ColDetectFieldEnabled=True; Kuka.CurrentCDSetIndex=0; Kuka.MovementParameterFieldEnabled=True; IlfCommand=SLIN
;ENDFOLD
SLIN XP326 WITH $VEL = SVEL_CP(2.0, , LCPDAT326),$TOOL = STOOL2(FP326),$BASE = SBASE(FP326.BASE_NO),$IPO_MODE = SIPO_MODE(FP326.IPO_FRAME),$LOAD = SLOAD(FP326.TOOL_NO),$ACC = SACC_CP(LCPDAT326),$ORI_TYPE = SORI_TYP(LCPDAT326),$APO = SAPO(LCPDAT326),$JERK = SJERK(LCPDAT326),$COLLMON_TOL_PRO[1] = USE_CM_PRO_VALUES(0)
;ENDFOLD

;FOLD SLIN P327 Vel=1 m/s CPDAT327 Tool[4]:Microflown3D Base[0];%{PE}
;FOLD Parameters ;%{h}
;Params IlfProvider=kukaroboter.basistech.inlineforms.movement.spline; Kuka.IsGlobalPoint=False; Kuka.PointName=P327; Kuka.BlendingEnabled=False; Kuka.MoveDataName=CPDAT327; Kuka.VelocityPath=1.000; Kuka.VelocityFieldEnabled=True; Kuka.ColDetectFieldEnabled=True; Kuka.CurrentCDSetIndex=0; Kuka.MovementParameterFieldEnabled=True; IlfCommand=SLIN
;ENDFOLD
SLIN XP327 WITH $VEL = SVEL_CP(2.0, , LCPDAT327),$TOOL = STOOL2(FP327),$BASE = SBASE(FP327.BASE_NO),$IPO_MODE = SIPO_MODE(FP327.IPO_FRAME),$LOAD = SLOAD(FP327.TOOL_NO),$ACC = SACC_CP(LCPDAT327),$ORI_TYPE = SORI_TYP(LCPDAT327),$APO = SAPO(LCPDAT327),$JERK = SJERK(LCPDAT327),$COLLMON_TOL_PRO[1] = USE_CM_PRO_VALUES(0)
;ENDFOLD

;FOLD SLIN P328 Vel=1 m/s CPDAT328 Tool[4]:Microflown3D Base[0];%{PE}
;FOLD Parameters ;%{h}
;Params IlfProvider=kukaroboter.basistech.inlineforms.movement.spline; Kuka.IsGlobalPoint=False; Kuka.PointName=P328; Kuka.BlendingEnabled=False; Kuka.MoveDataName=CPDAT328; Kuka.VelocityPath=1.000; Kuka.VelocityFieldEnabled=True; Kuka.ColDetectFieldEnabled=True; Kuka.CurrentCDSetIndex=0; Kuka.MovementParameterFieldEnabled=True; IlfCommand=SLIN
;ENDFOLD
SLIN XP328 WITH $VEL = SVEL_CP(2.0, , LCPDAT328),$TOOL = STOOL2(FP328),$BASE = SBASE(FP328.BASE_NO),$IPO_MODE = SIPO_MODE(FP328.IPO_FRAME),$LOAD = SLOAD(FP328.TOOL_NO),$ACC = SACC_CP(LCPDAT328),$ORI_TYPE = SORI_TYP(LCPDAT328),$APO = SAPO(LCPDAT328),$JERK = SJERK(LCPDAT328),$COLLMON_TOL_PRO[1] = USE_CM_PRO_VALUES(0)
;ENDFOLD

;FOLD SLIN P329 Vel=1 m/s CPDAT329 Tool[4]:Microflown3D Base[0];%{PE}
;FOLD Parameters ;%{h}
;Params IlfProvider=kukaroboter.basistech.inlineforms.movement.spline; Kuka.IsGlobalPoint=False; Kuka.PointName=P329; Kuka.BlendingEnabled=False; Kuka.MoveDataName=CPDAT329; Kuka.VelocityPath=1.000; Kuka.VelocityFieldEnabled=True; Kuka.ColDetectFieldEnabled=True; Kuka.CurrentCDSetIndex=0; Kuka.MovementParameterFieldEnabled=True; IlfCommand=SLIN
;ENDFOLD
SLIN XP329 WITH $VEL = SVEL_CP(2.0, , LCPDAT329),$TOOL = STOOL2(FP329),$BASE = SBASE(FP329.BASE_NO),$IPO_MODE = SIPO_MODE(FP329.IPO_FRAME),$LOAD = SLOAD(FP329.TOOL_NO),$ACC = SACC_CP(LCPDAT329),$ORI_TYPE = SORI_TYP(LCPDAT329),$APO = SAPO(LCPDAT329),$JERK = SJERK(LCPDAT329),$COLLMON_TOL_PRO[1] = USE_CM_PRO_VALUES(0)
;ENDFOLD

;FOLD SLIN P330 Vel=1 m/s CPDAT330 Tool[4]:Microflown3D Base[0];%{PE}
;FOLD Parameters ;%{h}
;Params IlfProvider=kukaroboter.basistech.inlineforms.movement.spline; Kuka.IsGlobalPoint=False; Kuka.PointName=P330; Kuka.BlendingEnabled=False; Kuka.MoveDataName=CPDAT330; Kuka.VelocityPath=1.000; Kuka.VelocityFieldEnabled=True; Kuka.ColDetectFieldEnabled=True; Kuka.CurrentCDSetIndex=0; Kuka.MovementParameterFieldEnabled=True; IlfCommand=SLIN
;ENDFOLD
SLIN XP330 WITH $VEL = SVEL_CP(2.0, , LCPDAT330),$TOOL = STOOL2(FP330),$BASE = SBASE(FP330.BASE_NO),$IPO_MODE = SIPO_MODE(FP330.IPO_FRAME),$LOAD = SLOAD(FP330.TOOL_NO),$ACC = SACC_CP(LCPDAT330),$ORI_TYPE = SORI_TYP(LCPDAT330),$APO = SAPO(LCPDAT330),$JERK = SJERK(LCPDAT330),$COLLMON_TOL_PRO[1] = USE_CM_PRO_VALUES(0)
;ENDFOLD

;FOLD SLIN P331 Vel=1 m/s CPDAT331 Tool[4]:Microflown3D Base[0];%{PE}
;FOLD Parameters ;%{h}
;Params IlfProvider=kukaroboter.basistech.inlineforms.movement.spline; Kuka.IsGlobalPoint=False; Kuka.PointName=P331; Kuka.BlendingEnabled=False; Kuka.MoveDataName=CPDAT331; Kuka.VelocityPath=1.000; Kuka.VelocityFieldEnabled=True; Kuka.ColDetectFieldEnabled=True; Kuka.CurrentCDSetIndex=0; Kuka.MovementParameterFieldEnabled=True; IlfCommand=SLIN
;ENDFOLD
SLIN XP331 WITH $VEL = SVEL_CP(2.0, , LCPDAT331),$TOOL = STOOL2(FP331),$BASE = SBASE(FP331.BASE_NO),$IPO_MODE = SIPO_MODE(FP331.IPO_FRAME),$LOAD = SLOAD(FP331.TOOL_NO),$ACC = SACC_CP(LCPDAT331),$ORI_TYPE = SORI_TYP(LCPDAT331),$APO = SAPO(LCPDAT331),$JERK = SJERK(LCPDAT331),$COLLMON_TOL_PRO[1] = USE_CM_PRO_VALUES(0)
;ENDFOLD

;FOLD SLIN P332 Vel=1 m/s CPDAT332 Tool[4]:Microflown3D Base[0];%{PE}
;FOLD Parameters ;%{h}
;Params IlfProvider=kukaroboter.basistech.inlineforms.movement.spline; Kuka.IsGlobalPoint=False; Kuka.PointName=P332; Kuka.BlendingEnabled=False; Kuka.MoveDataName=CPDAT332; Kuka.VelocityPath=1.000; Kuka.VelocityFieldEnabled=True; Kuka.ColDetectFieldEnabled=True; Kuka.CurrentCDSetIndex=0; Kuka.MovementParameterFieldEnabled=True; IlfCommand=SLIN
;ENDFOLD
SLIN XP332 WITH $VEL = SVEL_CP(2.0, , LCPDAT332),$TOOL = STOOL2(FP332),$BASE = SBASE(FP332.BASE_NO),$IPO_MODE = SIPO_MODE(FP332.IPO_FRAME),$LOAD = SLOAD(FP332.TOOL_NO),$ACC = SACC_CP(LCPDAT332),$ORI_TYPE = SORI_TYP(LCPDAT332),$APO = SAPO(LCPDAT332),$JERK = SJERK(LCPDAT332),$COLLMON_TOL_PRO[1] = USE_CM_PRO_VALUES(0)
;ENDFOLD

;FOLD SLIN P333 Vel=1 m/s CPDAT333 Tool[4]:Microflown3D Base[0];%{PE}
;FOLD Parameters ;%{h}
;Params IlfProvider=kukaroboter.basistech.inlineforms.movement.spline; Kuka.IsGlobalPoint=False; Kuka.PointName=P333; Kuka.BlendingEnabled=False; Kuka.MoveDataName=CPDAT333; Kuka.VelocityPath=1.000; Kuka.VelocityFieldEnabled=True; Kuka.ColDetectFieldEnabled=True; Kuka.CurrentCDSetIndex=0; Kuka.MovementParameterFieldEnabled=True; IlfCommand=SLIN
;ENDFOLD
SLIN XP333 WITH $VEL = SVEL_CP(2.0, , LCPDAT333),$TOOL = STOOL2(FP333),$BASE = SBASE(FP333.BASE_NO),$IPO_MODE = SIPO_MODE(FP333.IPO_FRAME),$LOAD = SLOAD(FP333.TOOL_NO),$ACC = SACC_CP(LCPDAT333),$ORI_TYPE = SORI_TYP(LCPDAT333),$APO = SAPO(LCPDAT333),$JERK = SJERK(LCPDAT333),$COLLMON_TOL_PRO[1] = USE_CM_PRO_VALUES(0)
;ENDFOLD

;FOLD SLIN P334 Vel=1 m/s CPDAT334 Tool[4]:Microflown3D Base[0];%{PE}
;FOLD Parameters ;%{h}
;Params IlfProvider=kukaroboter.basistech.inlineforms.movement.spline; Kuka.IsGlobalPoint=False; Kuka.PointName=P334; Kuka.BlendingEnabled=False; Kuka.MoveDataName=CPDAT334; Kuka.VelocityPath=1.000; Kuka.VelocityFieldEnabled=True; Kuka.ColDetectFieldEnabled=True; Kuka.CurrentCDSetIndex=0; Kuka.MovementParameterFieldEnabled=True; IlfCommand=SLIN
;ENDFOLD
SLIN XP334 WITH $VEL = SVEL_CP(2.0, , LCPDAT334),$TOOL = STOOL2(FP334),$BASE = SBASE(FP334.BASE_NO),$IPO_MODE = SIPO_MODE(FP334.IPO_FRAME),$LOAD = SLOAD(FP334.TOOL_NO),$ACC = SACC_CP(LCPDAT334),$ORI_TYPE = SORI_TYP(LCPDAT334),$APO = SAPO(LCPDAT334),$JERK = SJERK(LCPDAT334),$COLLMON_TOL_PRO[1] = USE_CM_PRO_VALUES(0)
;ENDFOLD

;FOLD SLIN P335 Vel=1 m/s CPDAT335 Tool[4]:Microflown3D Base[0];%{PE}
;FOLD Parameters ;%{h}
;Params IlfProvider=kukaroboter.basistech.inlineforms.movement.spline; Kuka.IsGlobalPoint=False; Kuka.PointName=P335; Kuka.BlendingEnabled=False; Kuka.MoveDataName=CPDAT335; Kuka.VelocityPath=1.000; Kuka.VelocityFieldEnabled=True; Kuka.ColDetectFieldEnabled=True; Kuka.CurrentCDSetIndex=0; Kuka.MovementParameterFieldEnabled=True; IlfCommand=SLIN
;ENDFOLD
SLIN XP335 WITH $VEL = SVEL_CP(2.0, , LCPDAT335),$TOOL = STOOL2(FP335),$BASE = SBASE(FP335.BASE_NO),$IPO_MODE = SIPO_MODE(FP335.IPO_FRAME),$LOAD = SLOAD(FP335.TOOL_NO),$ACC = SACC_CP(LCPDAT335),$ORI_TYPE = SORI_TYP(LCPDAT335),$APO = SAPO(LCPDAT335),$JERK = SJERK(LCPDAT335),$COLLMON_TOL_PRO[1] = USE_CM_PRO_VALUES(0)
;ENDFOLD

;FOLD SLIN P336 Vel=1 m/s CPDAT336 Tool[4]:Microflown3D Base[0];%{PE}
;FOLD Parameters ;%{h}
;Params IlfProvider=kukaroboter.basistech.inlineforms.movement.spline; Kuka.IsGlobalPoint=False; Kuka.PointName=P336; Kuka.BlendingEnabled=False; Kuka.MoveDataName=CPDAT336; Kuka.VelocityPath=1.000; Kuka.VelocityFieldEnabled=True; Kuka.ColDetectFieldEnabled=True; Kuka.CurrentCDSetIndex=0; Kuka.MovementParameterFieldEnabled=True; IlfCommand=SLIN
;ENDFOLD
SLIN XP336 WITH $VEL = SVEL_CP(2.0, , LCPDAT336),$TOOL = STOOL2(FP336),$BASE = SBASE(FP336.BASE_NO),$IPO_MODE = SIPO_MODE(FP336.IPO_FRAME),$LOAD = SLOAD(FP336.TOOL_NO),$ACC = SACC_CP(LCPDAT336),$ORI_TYPE = SORI_TYP(LCPDAT336),$APO = SAPO(LCPDAT336),$JERK = SJERK(LCPDAT336),$COLLMON_TOL_PRO[1] = USE_CM_PRO_VALUES(0)
;ENDFOLD

;FOLD SLIN P337 Vel=1 m/s CPDAT337 Tool[4]:Microflown3D Base[0];%{PE}
;FOLD Parameters ;%{h}
;Params IlfProvider=kukaroboter.basistech.inlineforms.movement.spline; Kuka.IsGlobalPoint=False; Kuka.PointName=P337; Kuka.BlendingEnabled=False; Kuka.MoveDataName=CPDAT337; Kuka.VelocityPath=1.000; Kuka.VelocityFieldEnabled=True; Kuka.ColDetectFieldEnabled=True; Kuka.CurrentCDSetIndex=0; Kuka.MovementParameterFieldEnabled=True; IlfCommand=SLIN
;ENDFOLD
SLIN XP337 WITH $VEL = SVEL_CP(2.0, , LCPDAT337),$TOOL = STOOL2(FP337),$BASE = SBASE(FP337.BASE_NO),$IPO_MODE = SIPO_MODE(FP337.IPO_FRAME),$LOAD = SLOAD(FP337.TOOL_NO),$ACC = SACC_CP(LCPDAT337),$ORI_TYPE = SORI_TYP(LCPDAT337),$APO = SAPO(LCPDAT337),$JERK = SJERK(LCPDAT337),$COLLMON_TOL_PRO[1] = USE_CM_PRO_VALUES(0)
;ENDFOLD

;FOLD SLIN P338 Vel=1 m/s CPDAT338 Tool[4]:Microflown3D Base[0];%{PE}
;FOLD Parameters ;%{h}
;Params IlfProvider=kukaroboter.basistech.inlineforms.movement.spline; Kuka.IsGlobalPoint=False; Kuka.PointName=P338; Kuka.BlendingEnabled=False; Kuka.MoveDataName=CPDAT338; Kuka.VelocityPath=1.000; Kuka.VelocityFieldEnabled=True; Kuka.ColDetectFieldEnabled=True; Kuka.CurrentCDSetIndex=0; Kuka.MovementParameterFieldEnabled=True; IlfCommand=SLIN
;ENDFOLD
SLIN XP338 WITH $VEL = SVEL_CP(2.0, , LCPDAT338),$TOOL = STOOL2(FP338),$BASE = SBASE(FP338.BASE_NO),$IPO_MODE = SIPO_MODE(FP338.IPO_FRAME),$LOAD = SLOAD(FP338.TOOL_NO),$ACC = SACC_CP(LCPDAT338),$ORI_TYPE = SORI_TYP(LCPDAT338),$APO = SAPO(LCPDAT338),$JERK = SJERK(LCPDAT338),$COLLMON_TOL_PRO[1] = USE_CM_PRO_VALUES(0)
;ENDFOLD

;FOLD SLIN P339 Vel=1 m/s CPDAT339 Tool[4]:Microflown3D Base[0];%{PE}
;FOLD Parameters ;%{h}
;Params IlfProvider=kukaroboter.basistech.inlineforms.movement.spline; Kuka.IsGlobalPoint=False; Kuka.PointName=P339; Kuka.BlendingEnabled=False; Kuka.MoveDataName=CPDAT339; Kuka.VelocityPath=1.000; Kuka.VelocityFieldEnabled=True; Kuka.ColDetectFieldEnabled=True; Kuka.CurrentCDSetIndex=0; Kuka.MovementParameterFieldEnabled=True; IlfCommand=SLIN
;ENDFOLD
SLIN XP339 WITH $VEL = SVEL_CP(2.0, , LCPDAT339),$TOOL = STOOL2(FP339),$BASE = SBASE(FP339.BASE_NO),$IPO_MODE = SIPO_MODE(FP339.IPO_FRAME),$LOAD = SLOAD(FP339.TOOL_NO),$ACC = SACC_CP(LCPDAT339),$ORI_TYPE = SORI_TYP(LCPDAT339),$APO = SAPO(LCPDAT339),$JERK = SJERK(LCPDAT339),$COLLMON_TOL_PRO[1] = USE_CM_PRO_VALUES(0)
;ENDFOLD

;FOLD SLIN P340 Vel=1 m/s CPDAT340 Tool[4]:Microflown3D Base[0];%{PE}
;FOLD Parameters ;%{h}
;Params IlfProvider=kukaroboter.basistech.inlineforms.movement.spline; Kuka.IsGlobalPoint=False; Kuka.PointName=P340; Kuka.BlendingEnabled=False; Kuka.MoveDataName=CPDAT340; Kuka.VelocityPath=1.000; Kuka.VelocityFieldEnabled=True; Kuka.ColDetectFieldEnabled=True; Kuka.CurrentCDSetIndex=0; Kuka.MovementParameterFieldEnabled=True; IlfCommand=SLIN
;ENDFOLD
SLIN XP340 WITH $VEL = SVEL_CP(2.0, , LCPDAT340),$TOOL = STOOL2(FP340),$BASE = SBASE(FP340.BASE_NO),$IPO_MODE = SIPO_MODE(FP340.IPO_FRAME),$LOAD = SLOAD(FP340.TOOL_NO),$ACC = SACC_CP(LCPDAT340),$ORI_TYPE = SORI_TYP(LCPDAT340),$APO = SAPO(LCPDAT340),$JERK = SJERK(LCPDAT340),$COLLMON_TOL_PRO[1] = USE_CM_PRO_VALUES(0)
;ENDFOLD

;FOLD SLIN P341 Vel=1 m/s CPDAT341 Tool[4]:Microflown3D Base[0];%{PE}
;FOLD Parameters ;%{h}
;Params IlfProvider=kukaroboter.basistech.inlineforms.movement.spline; Kuka.IsGlobalPoint=False; Kuka.PointName=P341; Kuka.BlendingEnabled=False; Kuka.MoveDataName=CPDAT341; Kuka.VelocityPath=1.000; Kuka.VelocityFieldEnabled=True; Kuka.ColDetectFieldEnabled=True; Kuka.CurrentCDSetIndex=0; Kuka.MovementParameterFieldEnabled=True; IlfCommand=SLIN
;ENDFOLD
SLIN XP341 WITH $VEL = SVEL_CP(2.0, , LCPDAT341),$TOOL = STOOL2(FP341),$BASE = SBASE(FP341.BASE_NO),$IPO_MODE = SIPO_MODE(FP341.IPO_FRAME),$LOAD = SLOAD(FP341.TOOL_NO),$ACC = SACC_CP(LCPDAT341),$ORI_TYPE = SORI_TYP(LCPDAT341),$APO = SAPO(LCPDAT341),$JERK = SJERK(LCPDAT341),$COLLMON_TOL_PRO[1] = USE_CM_PRO_VALUES(0)
;ENDFOLD

;FOLD SLIN P342 Vel=1 m/s CPDAT342 Tool[4]:Microflown3D Base[0];%{PE}
;FOLD Parameters ;%{h}
;Params IlfProvider=kukaroboter.basistech.inlineforms.movement.spline; Kuka.IsGlobalPoint=False; Kuka.PointName=P342; Kuka.BlendingEnabled=False; Kuka.MoveDataName=CPDAT342; Kuka.VelocityPath=1.000; Kuka.VelocityFieldEnabled=True; Kuka.ColDetectFieldEnabled=True; Kuka.CurrentCDSetIndex=0; Kuka.MovementParameterFieldEnabled=True; IlfCommand=SLIN
;ENDFOLD
SLIN XP342 WITH $VEL = SVEL_CP(2.0, , LCPDAT342),$TOOL = STOOL2(FP342),$BASE = SBASE(FP342.BASE_NO),$IPO_MODE = SIPO_MODE(FP342.IPO_FRAME),$LOAD = SLOAD(FP342.TOOL_NO),$ACC = SACC_CP(LCPDAT342),$ORI_TYPE = SORI_TYP(LCPDAT342),$APO = SAPO(LCPDAT342),$JERK = SJERK(LCPDAT342),$COLLMON_TOL_PRO[1] = USE_CM_PRO_VALUES(0)
;ENDFOLD

;FOLD SLIN P343 Vel=1 m/s CPDAT343 Tool[4]:Microflown3D Base[0];%{PE}
;FOLD Parameters ;%{h}
;Params IlfProvider=kukaroboter.basistech.inlineforms.movement.spline; Kuka.IsGlobalPoint=False; Kuka.PointName=P343; Kuka.BlendingEnabled=False; Kuka.MoveDataName=CPDAT343; Kuka.VelocityPath=1.000; Kuka.VelocityFieldEnabled=True; Kuka.ColDetectFieldEnabled=True; Kuka.CurrentCDSetIndex=0; Kuka.MovementParameterFieldEnabled=True; IlfCommand=SLIN
;ENDFOLD
SLIN XP343 WITH $VEL = SVEL_CP(2.0, , LCPDAT343),$TOOL = STOOL2(FP343),$BASE = SBASE(FP343.BASE_NO),$IPO_MODE = SIPO_MODE(FP343.IPO_FRAME),$LOAD = SLOAD(FP343.TOOL_NO),$ACC = SACC_CP(LCPDAT343),$ORI_TYPE = SORI_TYP(LCPDAT343),$APO = SAPO(LCPDAT343),$JERK = SJERK(LCPDAT343),$COLLMON_TOL_PRO[1] = USE_CM_PRO_VALUES(0)
;ENDFOLD

;FOLD SLIN P344 Vel=1 m/s CPDAT344 Tool[4]:Microflown3D Base[0];%{PE}
;FOLD Parameters ;%{h}
;Params IlfProvider=kukaroboter.basistech.inlineforms.movement.spline; Kuka.IsGlobalPoint=False; Kuka.PointName=P344; Kuka.BlendingEnabled=False; Kuka.MoveDataName=CPDAT344; Kuka.VelocityPath=1.000; Kuka.VelocityFieldEnabled=True; Kuka.ColDetectFieldEnabled=True; Kuka.CurrentCDSetIndex=0; Kuka.MovementParameterFieldEnabled=True; IlfCommand=SLIN
;ENDFOLD
SLIN XP344 WITH $VEL = SVEL_CP(2.0, , LCPDAT344),$TOOL = STOOL2(FP344),$BASE = SBASE(FP344.BASE_NO),$IPO_MODE = SIPO_MODE(FP344.IPO_FRAME),$LOAD = SLOAD(FP344.TOOL_NO),$ACC = SACC_CP(LCPDAT344),$ORI_TYPE = SORI_TYP(LCPDAT344),$APO = SAPO(LCPDAT344),$JERK = SJERK(LCPDAT344),$COLLMON_TOL_PRO[1] = USE_CM_PRO_VALUES(0)
;ENDFOLD

;FOLD SLIN P345 Vel=1 m/s CPDAT345 Tool[4]:Microflown3D Base[0];%{PE}
;FOLD Parameters ;%{h}
;Params IlfProvider=kukaroboter.basistech.inlineforms.movement.spline; Kuka.IsGlobalPoint=False; Kuka.PointName=P345; Kuka.BlendingEnabled=False; Kuka.MoveDataName=CPDAT345; Kuka.VelocityPath=1.000; Kuka.VelocityFieldEnabled=True; Kuka.ColDetectFieldEnabled=True; Kuka.CurrentCDSetIndex=0; Kuka.MovementParameterFieldEnabled=True; IlfCommand=SLIN
;ENDFOLD
SLIN XP345 WITH $VEL = SVEL_CP(2.0, , LCPDAT345),$TOOL = STOOL2(FP345),$BASE = SBASE(FP345.BASE_NO),$IPO_MODE = SIPO_MODE(FP345.IPO_FRAME),$LOAD = SLOAD(FP345.TOOL_NO),$ACC = SACC_CP(LCPDAT345),$ORI_TYPE = SORI_TYP(LCPDAT345),$APO = SAPO(LCPDAT345),$JERK = SJERK(LCPDAT345),$COLLMON_TOL_PRO[1] = USE_CM_PRO_VALUES(0)
;ENDFOLD

;FOLD SLIN P346 Vel=1 m/s CPDAT346 Tool[4]:Microflown3D Base[0];%{PE}
;FOLD Parameters ;%{h}
;Params IlfProvider=kukaroboter.basistech.inlineforms.movement.spline; Kuka.IsGlobalPoint=False; Kuka.PointName=P346; Kuka.BlendingEnabled=False; Kuka.MoveDataName=CPDAT346; Kuka.VelocityPath=1.000; Kuka.VelocityFieldEnabled=True; Kuka.ColDetectFieldEnabled=True; Kuka.CurrentCDSetIndex=0; Kuka.MovementParameterFieldEnabled=True; IlfCommand=SLIN
;ENDFOLD
SLIN XP346 WITH $VEL = SVEL_CP(2.0, , LCPDAT346),$TOOL = STOOL2(FP346),$BASE = SBASE(FP346.BASE_NO),$IPO_MODE = SIPO_MODE(FP346.IPO_FRAME),$LOAD = SLOAD(FP346.TOOL_NO),$ACC = SACC_CP(LCPDAT346),$ORI_TYPE = SORI_TYP(LCPDAT346),$APO = SAPO(LCPDAT346),$JERK = SJERK(LCPDAT346),$COLLMON_TOL_PRO[1] = USE_CM_PRO_VALUES(0)
;ENDFOLD

;FOLD SLIN P347 Vel=1 m/s CPDAT347 Tool[4]:Microflown3D Base[0];%{PE}
;FOLD Parameters ;%{h}
;Params IlfProvider=kukaroboter.basistech.inlineforms.movement.spline; Kuka.IsGlobalPoint=False; Kuka.PointName=P347; Kuka.BlendingEnabled=False; Kuka.MoveDataName=CPDAT347; Kuka.VelocityPath=1.000; Kuka.VelocityFieldEnabled=True; Kuka.ColDetectFieldEnabled=True; Kuka.CurrentCDSetIndex=0; Kuka.MovementParameterFieldEnabled=True; IlfCommand=SLIN
;ENDFOLD
SLIN XP347 WITH $VEL = SVEL_CP(2.0, , LCPDAT347),$TOOL = STOOL2(FP347),$BASE = SBASE(FP347.BASE_NO),$IPO_MODE = SIPO_MODE(FP347.IPO_FRAME),$LOAD = SLOAD(FP347.TOOL_NO),$ACC = SACC_CP(LCPDAT347),$ORI_TYPE = SORI_TYP(LCPDAT347),$APO = SAPO(LCPDAT347),$JERK = SJERK(LCPDAT347),$COLLMON_TOL_PRO[1] = USE_CM_PRO_VALUES(0)
;ENDFOLD

;FOLD SLIN P348 Vel=1 m/s CPDAT348 Tool[4]:Microflown3D Base[0];%{PE}
;FOLD Parameters ;%{h}
;Params IlfProvider=kukaroboter.basistech.inlineforms.movement.spline; Kuka.IsGlobalPoint=False; Kuka.PointName=P348; Kuka.BlendingEnabled=False; Kuka.MoveDataName=CPDAT348; Kuka.VelocityPath=1.000; Kuka.VelocityFieldEnabled=True; Kuka.ColDetectFieldEnabled=True; Kuka.CurrentCDSetIndex=0; Kuka.MovementParameterFieldEnabled=True; IlfCommand=SLIN
;ENDFOLD
SLIN XP348 WITH $VEL = SVEL_CP(2.0, , LCPDAT348),$TOOL = STOOL2(FP348),$BASE = SBASE(FP348.BASE_NO),$IPO_MODE = SIPO_MODE(FP348.IPO_FRAME),$LOAD = SLOAD(FP348.TOOL_NO),$ACC = SACC_CP(LCPDAT348),$ORI_TYPE = SORI_TYP(LCPDAT348),$APO = SAPO(LCPDAT348),$JERK = SJERK(LCPDAT348),$COLLMON_TOL_PRO[1] = USE_CM_PRO_VALUES(0)
;ENDFOLD

;FOLD SLIN P349 Vel=1 m/s CPDAT349 Tool[4]:Microflown3D Base[0];%{PE}
;FOLD Parameters ;%{h}
;Params IlfProvider=kukaroboter.basistech.inlineforms.movement.spline; Kuka.IsGlobalPoint=False; Kuka.PointName=P349; Kuka.BlendingEnabled=False; Kuka.MoveDataName=CPDAT349; Kuka.VelocityPath=1.000; Kuka.VelocityFieldEnabled=True; Kuka.ColDetectFieldEnabled=True; Kuka.CurrentCDSetIndex=0; Kuka.MovementParameterFieldEnabled=True; IlfCommand=SLIN
;ENDFOLD
SLIN XP349 WITH $VEL = SVEL_CP(2.0, , LCPDAT349),$TOOL = STOOL2(FP349),$BASE = SBASE(FP349.BASE_NO),$IPO_MODE = SIPO_MODE(FP349.IPO_FRAME),$LOAD = SLOAD(FP349.TOOL_NO),$ACC = SACC_CP(LCPDAT349),$ORI_TYPE = SORI_TYP(LCPDAT349),$APO = SAPO(LCPDAT349),$JERK = SJERK(LCPDAT349),$COLLMON_TOL_PRO[1] = USE_CM_PRO_VALUES(0)
;ENDFOLD

;FOLD SLIN P350 Vel=1 m/s CPDAT350 Tool[4]:Microflown3D Base[0];%{PE}
;FOLD Parameters ;%{h}
;Params IlfProvider=kukaroboter.basistech.inlineforms.movement.spline; Kuka.IsGlobalPoint=False; Kuka.PointName=P350; Kuka.BlendingEnabled=False; Kuka.MoveDataName=CPDAT350; Kuka.VelocityPath=1.000; Kuka.VelocityFieldEnabled=True; Kuka.ColDetectFieldEnabled=True; Kuka.CurrentCDSetIndex=0; Kuka.MovementParameterFieldEnabled=True; IlfCommand=SLIN
;ENDFOLD
SLIN XP350 WITH $VEL = SVEL_CP(2.0, , LCPDAT350),$TOOL = STOOL2(FP350),$BASE = SBASE(FP350.BASE_NO),$IPO_MODE = SIPO_MODE(FP350.IPO_FRAME),$LOAD = SLOAD(FP350.TOOL_NO),$ACC = SACC_CP(LCPDAT350),$ORI_TYPE = SORI_TYP(LCPDAT350),$APO = SAPO(LCPDAT350),$JERK = SJERK(LCPDAT350),$COLLMON_TOL_PRO[1] = USE_CM_PRO_VALUES(0)
;ENDFOLD

;FOLD SLIN P351 Vel=1 m/s CPDAT351 Tool[4]:Microflown3D Base[0];%{PE}
;FOLD Parameters ;%{h}
;Params IlfProvider=kukaroboter.basistech.inlineforms.movement.spline; Kuka.IsGlobalPoint=False; Kuka.PointName=P351; Kuka.BlendingEnabled=False; Kuka.MoveDataName=CPDAT351; Kuka.VelocityPath=1.000; Kuka.VelocityFieldEnabled=True; Kuka.ColDetectFieldEnabled=True; Kuka.CurrentCDSetIndex=0; Kuka.MovementParameterFieldEnabled=True; IlfCommand=SLIN
;ENDFOLD
SLIN XP351 WITH $VEL = SVEL_CP(2.0, , LCPDAT351),$TOOL = STOOL2(FP351),$BASE = SBASE(FP351.BASE_NO),$IPO_MODE = SIPO_MODE(FP351.IPO_FRAME),$LOAD = SLOAD(FP351.TOOL_NO),$ACC = SACC_CP(LCPDAT351),$ORI_TYPE = SORI_TYP(LCPDAT351),$APO = SAPO(LCPDAT351),$JERK = SJERK(LCPDAT351),$COLLMON_TOL_PRO[1] = USE_CM_PRO_VALUES(0)
;ENDFOLD

;FOLD SLIN P352 Vel=1 m/s CPDAT352 Tool[4]:Microflown3D Base[0];%{PE}
;FOLD Parameters ;%{h}
;Params IlfProvider=kukaroboter.basistech.inlineforms.movement.spline; Kuka.IsGlobalPoint=False; Kuka.PointName=P352; Kuka.BlendingEnabled=False; Kuka.MoveDataName=CPDAT352; Kuka.VelocityPath=1.000; Kuka.VelocityFieldEnabled=True; Kuka.ColDetectFieldEnabled=True; Kuka.CurrentCDSetIndex=0; Kuka.MovementParameterFieldEnabled=True; IlfCommand=SLIN
;ENDFOLD
SLIN XP352 WITH $VEL = SVEL_CP(2.0, , LCPDAT352),$TOOL = STOOL2(FP352),$BASE = SBASE(FP352.BASE_NO),$IPO_MODE = SIPO_MODE(FP352.IPO_FRAME),$LOAD = SLOAD(FP352.TOOL_NO),$ACC = SACC_CP(LCPDAT352),$ORI_TYPE = SORI_TYP(LCPDAT352),$APO = SAPO(LCPDAT352),$JERK = SJERK(LCPDAT352),$COLLMON_TOL_PRO[1] = USE_CM_PRO_VALUES(0)
;ENDFOLD

;FOLD SLIN P353 Vel=1 m/s CPDAT353 Tool[4]:Microflown3D Base[0];%{PE}
;FOLD Parameters ;%{h}
;Params IlfProvider=kukaroboter.basistech.inlineforms.movement.spline; Kuka.IsGlobalPoint=False; Kuka.PointName=P353; Kuka.BlendingEnabled=False; Kuka.MoveDataName=CPDAT353; Kuka.VelocityPath=1.000; Kuka.VelocityFieldEnabled=True; Kuka.ColDetectFieldEnabled=True; Kuka.CurrentCDSetIndex=0; Kuka.MovementParameterFieldEnabled=True; IlfCommand=SLIN
;ENDFOLD
SLIN XP353 WITH $VEL = SVEL_CP(2.0, , LCPDAT353),$TOOL = STOOL2(FP353),$BASE = SBASE(FP353.BASE_NO),$IPO_MODE = SIPO_MODE(FP353.IPO_FRAME),$LOAD = SLOAD(FP353.TOOL_NO),$ACC = SACC_CP(LCPDAT353),$ORI_TYPE = SORI_TYP(LCPDAT353),$APO = SAPO(LCPDAT353),$JERK = SJERK(LCPDAT353),$COLLMON_TOL_PRO[1] = USE_CM_PRO_VALUES(0)
;ENDFOLD

;FOLD SLIN P354 Vel=1 m/s CPDAT354 Tool[4]:Microflown3D Base[0];%{PE}
;FOLD Parameters ;%{h}
;Params IlfProvider=kukaroboter.basistech.inlineforms.movement.spline; Kuka.IsGlobalPoint=False; Kuka.PointName=P354; Kuka.BlendingEnabled=False; Kuka.MoveDataName=CPDAT354; Kuka.VelocityPath=1.000; Kuka.VelocityFieldEnabled=True; Kuka.ColDetectFieldEnabled=True; Kuka.CurrentCDSetIndex=0; Kuka.MovementParameterFieldEnabled=True; IlfCommand=SLIN
;ENDFOLD
SLIN XP354 WITH $VEL = SVEL_CP(2.0, , LCPDAT354),$TOOL = STOOL2(FP354),$BASE = SBASE(FP354.BASE_NO),$IPO_MODE = SIPO_MODE(FP354.IPO_FRAME),$LOAD = SLOAD(FP354.TOOL_NO),$ACC = SACC_CP(LCPDAT354),$ORI_TYPE = SORI_TYP(LCPDAT354),$APO = SAPO(LCPDAT354),$JERK = SJERK(LCPDAT354),$COLLMON_TOL_PRO[1] = USE_CM_PRO_VALUES(0)
;ENDFOLD

;FOLD SLIN P355 Vel=1 m/s CPDAT355 Tool[4]:Microflown3D Base[0];%{PE}
;FOLD Parameters ;%{h}
;Params IlfProvider=kukaroboter.basistech.inlineforms.movement.spline; Kuka.IsGlobalPoint=False; Kuka.PointName=P355; Kuka.BlendingEnabled=False; Kuka.MoveDataName=CPDAT355; Kuka.VelocityPath=1.000; Kuka.VelocityFieldEnabled=True; Kuka.ColDetectFieldEnabled=True; Kuka.CurrentCDSetIndex=0; Kuka.MovementParameterFieldEnabled=True; IlfCommand=SLIN
;ENDFOLD
SLIN XP355 WITH $VEL = SVEL_CP(2.0, , LCPDAT355),$TOOL = STOOL2(FP355),$BASE = SBASE(FP355.BASE_NO),$IPO_MODE = SIPO_MODE(FP355.IPO_FRAME),$LOAD = SLOAD(FP355.TOOL_NO),$ACC = SACC_CP(LCPDAT355),$ORI_TYPE = SORI_TYP(LCPDAT355),$APO = SAPO(LCPDAT355),$JERK = SJERK(LCPDAT355),$COLLMON_TOL_PRO[1] = USE_CM_PRO_VALUES(0)
;ENDFOLD

;FOLD SLIN P356 Vel=1 m/s CPDAT356 Tool[4]:Microflown3D Base[0];%{PE}
;FOLD Parameters ;%{h}
;Params IlfProvider=kukaroboter.basistech.inlineforms.movement.spline; Kuka.IsGlobalPoint=False; Kuka.PointName=P356; Kuka.BlendingEnabled=False; Kuka.MoveDataName=CPDAT356; Kuka.VelocityPath=1.000; Kuka.VelocityFieldEnabled=True; Kuka.ColDetectFieldEnabled=True; Kuka.CurrentCDSetIndex=0; Kuka.MovementParameterFieldEnabled=True; IlfCommand=SLIN
;ENDFOLD
SLIN XP356 WITH $VEL = SVEL_CP(2.0, , LCPDAT356),$TOOL = STOOL2(FP356),$BASE = SBASE(FP356.BASE_NO),$IPO_MODE = SIPO_MODE(FP356.IPO_FRAME),$LOAD = SLOAD(FP356.TOOL_NO),$ACC = SACC_CP(LCPDAT356),$ORI_TYPE = SORI_TYP(LCPDAT356),$APO = SAPO(LCPDAT356),$JERK = SJERK(LCPDAT356),$COLLMON_TOL_PRO[1] = USE_CM_PRO_VALUES(0)
;ENDFOLD

;FOLD SLIN P357 Vel=1 m/s CPDAT357 Tool[4]:Microflown3D Base[0];%{PE}
;FOLD Parameters ;%{h}
;Params IlfProvider=kukaroboter.basistech.inlineforms.movement.spline; Kuka.IsGlobalPoint=False; Kuka.PointName=P357; Kuka.BlendingEnabled=False; Kuka.MoveDataName=CPDAT357; Kuka.VelocityPath=1.000; Kuka.VelocityFieldEnabled=True; Kuka.ColDetectFieldEnabled=True; Kuka.CurrentCDSetIndex=0; Kuka.MovementParameterFieldEnabled=True; IlfCommand=SLIN
;ENDFOLD
SLIN XP357 WITH $VEL = SVEL_CP(2.0, , LCPDAT357),$TOOL = STOOL2(FP357),$BASE = SBASE(FP357.BASE_NO),$IPO_MODE = SIPO_MODE(FP357.IPO_FRAME),$LOAD = SLOAD(FP357.TOOL_NO),$ACC = SACC_CP(LCPDAT357),$ORI_TYPE = SORI_TYP(LCPDAT357),$APO = SAPO(LCPDAT357),$JERK = SJERK(LCPDAT357),$COLLMON_TOL_PRO[1] = USE_CM_PRO_VALUES(0)
;ENDFOLD

;FOLD SLIN P358 Vel=1 m/s CPDAT358 Tool[4]:Microflown3D Base[0];%{PE}
;FOLD Parameters ;%{h}
;Params IlfProvider=kukaroboter.basistech.inlineforms.movement.spline; Kuka.IsGlobalPoint=False; Kuka.PointName=P358; Kuka.BlendingEnabled=False; Kuka.MoveDataName=CPDAT358; Kuka.VelocityPath=1.000; Kuka.VelocityFieldEnabled=True; Kuka.ColDetectFieldEnabled=True; Kuka.CurrentCDSetIndex=0; Kuka.MovementParameterFieldEnabled=True; IlfCommand=SLIN
;ENDFOLD
SLIN XP358 WITH $VEL = SVEL_CP(2.0, , LCPDAT358),$TOOL = STOOL2(FP358),$BASE = SBASE(FP358.BASE_NO),$IPO_MODE = SIPO_MODE(FP358.IPO_FRAME),$LOAD = SLOAD(FP358.TOOL_NO),$ACC = SACC_CP(LCPDAT358),$ORI_TYPE = SORI_TYP(LCPDAT358),$APO = SAPO(LCPDAT358),$JERK = SJERK(LCPDAT358),$COLLMON_TOL_PRO[1] = USE_CM_PRO_VALUES(0)
;ENDFOLD

;FOLD SLIN P359 Vel=1 m/s CPDAT359 Tool[4]:Microflown3D Base[0];%{PE}
;FOLD Parameters ;%{h}
;Params IlfProvider=kukaroboter.basistech.inlineforms.movement.spline; Kuka.IsGlobalPoint=False; Kuka.PointName=P359; Kuka.BlendingEnabled=False; Kuka.MoveDataName=CPDAT359; Kuka.VelocityPath=1.000; Kuka.VelocityFieldEnabled=True; Kuka.ColDetectFieldEnabled=True; Kuka.CurrentCDSetIndex=0; Kuka.MovementParameterFieldEnabled=True; IlfCommand=SLIN
;ENDFOLD
SLIN XP359 WITH $VEL = SVEL_CP(2.0, , LCPDAT359),$TOOL = STOOL2(FP359),$BASE = SBASE(FP359.BASE_NO),$IPO_MODE = SIPO_MODE(FP359.IPO_FRAME),$LOAD = SLOAD(FP359.TOOL_NO),$ACC = SACC_CP(LCPDAT359),$ORI_TYPE = SORI_TYP(LCPDAT359),$APO = SAPO(LCPDAT359),$JERK = SJERK(LCPDAT359),$COLLMON_TOL_PRO[1] = USE_CM_PRO_VALUES(0)
;ENDFOLD

;FOLD SLIN P360 Vel=1 m/s CPDAT360 Tool[4]:Microflown3D Base[0];%{PE}
;FOLD Parameters ;%{h}
;Params IlfProvider=kukaroboter.basistech.inlineforms.movement.spline; Kuka.IsGlobalPoint=False; Kuka.PointName=P360; Kuka.BlendingEnabled=False; Kuka.MoveDataName=CPDAT360; Kuka.VelocityPath=1.000; Kuka.VelocityFieldEnabled=True; Kuka.ColDetectFieldEnabled=True; Kuka.CurrentCDSetIndex=0; Kuka.MovementParameterFieldEnabled=True; IlfCommand=SLIN
;ENDFOLD
SLIN XP360 WITH $VEL = SVEL_CP(2.0, , LCPDAT360),$TOOL = STOOL2(FP360),$BASE = SBASE(FP360.BASE_NO),$IPO_MODE = SIPO_MODE(FP360.IPO_FRAME),$LOAD = SLOAD(FP360.TOOL_NO),$ACC = SACC_CP(LCPDAT360),$ORI_TYPE = SORI_TYP(LCPDAT360),$APO = SAPO(LCPDAT360),$JERK = SJERK(LCPDAT360),$COLLMON_TOL_PRO[1] = USE_CM_PRO_VALUES(0)
;ENDFOLD

;FOLD SLIN P361 Vel=1 m/s CPDAT361 Tool[4]:Microflown3D Base[0];%{PE}
;FOLD Parameters ;%{h}
;Params IlfProvider=kukaroboter.basistech.inlineforms.movement.spline; Kuka.IsGlobalPoint=False; Kuka.PointName=P361; Kuka.BlendingEnabled=False; Kuka.MoveDataName=CPDAT361; Kuka.VelocityPath=1.000; Kuka.VelocityFieldEnabled=True; Kuka.ColDetectFieldEnabled=True; Kuka.CurrentCDSetIndex=0; Kuka.MovementParameterFieldEnabled=True; IlfCommand=SLIN
;ENDFOLD
SLIN XP361 WITH $VEL = SVEL_CP(2.0, , LCPDAT361),$TOOL = STOOL2(FP361),$BASE = SBASE(FP361.BASE_NO),$IPO_MODE = SIPO_MODE(FP361.IPO_FRAME),$LOAD = SLOAD(FP361.TOOL_NO),$ACC = SACC_CP(LCPDAT361),$ORI_TYPE = SORI_TYP(LCPDAT361),$APO = SAPO(LCPDAT361),$JERK = SJERK(LCPDAT361),$COLLMON_TOL_PRO[1] = USE_CM_PRO_VALUES(0)
;ENDFOLD

;FOLD SLIN P362 Vel=1 m/s CPDAT362 Tool[4]:Microflown3D Base[0];%{PE}
;FOLD Parameters ;%{h}
;Params IlfProvider=kukaroboter.basistech.inlineforms.movement.spline; Kuka.IsGlobalPoint=False; Kuka.PointName=P362; Kuka.BlendingEnabled=False; Kuka.MoveDataName=CPDAT362; Kuka.VelocityPath=1.000; Kuka.VelocityFieldEnabled=True; Kuka.ColDetectFieldEnabled=True; Kuka.CurrentCDSetIndex=0; Kuka.MovementParameterFieldEnabled=True; IlfCommand=SLIN
;ENDFOLD
SLIN XP362 WITH $VEL = SVEL_CP(2.0, , LCPDAT362),$TOOL = STOOL2(FP362),$BASE = SBASE(FP362.BASE_NO),$IPO_MODE = SIPO_MODE(FP362.IPO_FRAME),$LOAD = SLOAD(FP362.TOOL_NO),$ACC = SACC_CP(LCPDAT362),$ORI_TYPE = SORI_TYP(LCPDAT362),$APO = SAPO(LCPDAT362),$JERK = SJERK(LCPDAT362),$COLLMON_TOL_PRO[1] = USE_CM_PRO_VALUES(0)
;ENDFOLD

;FOLD SLIN P363 Vel=1 m/s CPDAT363 Tool[4]:Microflown3D Base[0];%{PE}
;FOLD Parameters ;%{h}
;Params IlfProvider=kukaroboter.basistech.inlineforms.movement.spline; Kuka.IsGlobalPoint=False; Kuka.PointName=P363; Kuka.BlendingEnabled=False; Kuka.MoveDataName=CPDAT363; Kuka.VelocityPath=1.000; Kuka.VelocityFieldEnabled=True; Kuka.ColDetectFieldEnabled=True; Kuka.CurrentCDSetIndex=0; Kuka.MovementParameterFieldEnabled=True; IlfCommand=SLIN
;ENDFOLD
SLIN XP363 WITH $VEL = SVEL_CP(2.0, , LCPDAT363),$TOOL = STOOL2(FP363),$BASE = SBASE(FP363.BASE_NO),$IPO_MODE = SIPO_MODE(FP363.IPO_FRAME),$LOAD = SLOAD(FP363.TOOL_NO),$ACC = SACC_CP(LCPDAT363),$ORI_TYPE = SORI_TYP(LCPDAT363),$APO = SAPO(LCPDAT363),$JERK = SJERK(LCPDAT363),$COLLMON_TOL_PRO[1] = USE_CM_PRO_VALUES(0)
;ENDFOLD

;FOLD SLIN P364 Vel=1 m/s CPDAT364 Tool[4]:Microflown3D Base[0];%{PE}
;FOLD Parameters ;%{h}
;Params IlfProvider=kukaroboter.basistech.inlineforms.movement.spline; Kuka.IsGlobalPoint=False; Kuka.PointName=P364; Kuka.BlendingEnabled=False; Kuka.MoveDataName=CPDAT364; Kuka.VelocityPath=1.000; Kuka.VelocityFieldEnabled=True; Kuka.ColDetectFieldEnabled=True; Kuka.CurrentCDSetIndex=0; Kuka.MovementParameterFieldEnabled=True; IlfCommand=SLIN
;ENDFOLD
SLIN XP364 WITH $VEL = SVEL_CP(2.0, , LCPDAT364),$TOOL = STOOL2(FP364),$BASE = SBASE(FP364.BASE_NO),$IPO_MODE = SIPO_MODE(FP364.IPO_FRAME),$LOAD = SLOAD(FP364.TOOL_NO),$ACC = SACC_CP(LCPDAT364),$ORI_TYPE = SORI_TYP(LCPDAT364),$APO = SAPO(LCPDAT364),$JERK = SJERK(LCPDAT364),$COLLMON_TOL_PRO[1] = USE_CM_PRO_VALUES(0)
;ENDFOLD

;FOLD SLIN P365 Vel=1 m/s CPDAT365 Tool[4]:Microflown3D Base[0];%{PE}
;FOLD Parameters ;%{h}
;Params IlfProvider=kukaroboter.basistech.inlineforms.movement.spline; Kuka.IsGlobalPoint=False; Kuka.PointName=P365; Kuka.BlendingEnabled=False; Kuka.MoveDataName=CPDAT365; Kuka.VelocityPath=1.000; Kuka.VelocityFieldEnabled=True; Kuka.ColDetectFieldEnabled=True; Kuka.CurrentCDSetIndex=0; Kuka.MovementParameterFieldEnabled=True; IlfCommand=SLIN
;ENDFOLD
SLIN XP365 WITH $VEL = SVEL_CP(2.0, , LCPDAT365),$TOOL = STOOL2(FP365),$BASE = SBASE(FP365.BASE_NO),$IPO_MODE = SIPO_MODE(FP365.IPO_FRAME),$LOAD = SLOAD(FP365.TOOL_NO),$ACC = SACC_CP(LCPDAT365),$ORI_TYPE = SORI_TYP(LCPDAT365),$APO = SAPO(LCPDAT365),$JERK = SJERK(LCPDAT365),$COLLMON_TOL_PRO[1] = USE_CM_PRO_VALUES(0)
;ENDFOLD

;FOLD SLIN P366 Vel=1 m/s CPDAT366 Tool[4]:Microflown3D Base[0];%{PE}
;FOLD Parameters ;%{h}
;Params IlfProvider=kukaroboter.basistech.inlineforms.movement.spline; Kuka.IsGlobalPoint=False; Kuka.PointName=P366; Kuka.BlendingEnabled=False; Kuka.MoveDataName=CPDAT366; Kuka.VelocityPath=1.000; Kuka.VelocityFieldEnabled=True; Kuka.ColDetectFieldEnabled=True; Kuka.CurrentCDSetIndex=0; Kuka.MovementParameterFieldEnabled=True; IlfCommand=SLIN
;ENDFOLD
SLIN XP366 WITH $VEL = SVEL_CP(2.0, , LCPDAT366),$TOOL = STOOL2(FP366),$BASE = SBASE(FP366.BASE_NO),$IPO_MODE = SIPO_MODE(FP366.IPO_FRAME),$LOAD = SLOAD(FP366.TOOL_NO),$ACC = SACC_CP(LCPDAT366),$ORI_TYPE = SORI_TYP(LCPDAT366),$APO = SAPO(LCPDAT366),$JERK = SJERK(LCPDAT366),$COLLMON_TOL_PRO[1] = USE_CM_PRO_VALUES(0)
;ENDFOLD

;FOLD SLIN P367 Vel=1 m/s CPDAT367 Tool[4]:Microflown3D Base[0];%{PE}
;FOLD Parameters ;%{h}
;Params IlfProvider=kukaroboter.basistech.inlineforms.movement.spline; Kuka.IsGlobalPoint=False; Kuka.PointName=P367; Kuka.BlendingEnabled=False; Kuka.MoveDataName=CPDAT367; Kuka.VelocityPath=1.000; Kuka.VelocityFieldEnabled=True; Kuka.ColDetectFieldEnabled=True; Kuka.CurrentCDSetIndex=0; Kuka.MovementParameterFieldEnabled=True; IlfCommand=SLIN
;ENDFOLD
SLIN XP367 WITH $VEL = SVEL_CP(2.0, , LCPDAT367),$TOOL = STOOL2(FP367),$BASE = SBASE(FP367.BASE_NO),$IPO_MODE = SIPO_MODE(FP367.IPO_FRAME),$LOAD = SLOAD(FP367.TOOL_NO),$ACC = SACC_CP(LCPDAT367),$ORI_TYPE = SORI_TYP(LCPDAT367),$APO = SAPO(LCPDAT367),$JERK = SJERK(LCPDAT367),$COLLMON_TOL_PRO[1] = USE_CM_PRO_VALUES(0)
;ENDFOLD

;FOLD SLIN P368 Vel=1 m/s CPDAT368 Tool[4]:Microflown3D Base[0];%{PE}
;FOLD Parameters ;%{h}
;Params IlfProvider=kukaroboter.basistech.inlineforms.movement.spline; Kuka.IsGlobalPoint=False; Kuka.PointName=P368; Kuka.BlendingEnabled=False; Kuka.MoveDataName=CPDAT368; Kuka.VelocityPath=1.000; Kuka.VelocityFieldEnabled=True; Kuka.ColDetectFieldEnabled=True; Kuka.CurrentCDSetIndex=0; Kuka.MovementParameterFieldEnabled=True; IlfCommand=SLIN
;ENDFOLD
SLIN XP368 WITH $VEL = SVEL_CP(2.0, , LCPDAT368),$TOOL = STOOL2(FP368),$BASE = SBASE(FP368.BASE_NO),$IPO_MODE = SIPO_MODE(FP368.IPO_FRAME),$LOAD = SLOAD(FP368.TOOL_NO),$ACC = SACC_CP(LCPDAT368),$ORI_TYPE = SORI_TYP(LCPDAT368),$APO = SAPO(LCPDAT368),$JERK = SJERK(LCPDAT368),$COLLMON_TOL_PRO[1] = USE_CM_PRO_VALUES(0)
;ENDFOLD

;FOLD SLIN P369 Vel=1 m/s CPDAT369 Tool[4]:Microflown3D Base[0];%{PE}
;FOLD Parameters ;%{h}
;Params IlfProvider=kukaroboter.basistech.inlineforms.movement.spline; Kuka.IsGlobalPoint=False; Kuka.PointName=P369; Kuka.BlendingEnabled=False; Kuka.MoveDataName=CPDAT369; Kuka.VelocityPath=1.000; Kuka.VelocityFieldEnabled=True; Kuka.ColDetectFieldEnabled=True; Kuka.CurrentCDSetIndex=0; Kuka.MovementParameterFieldEnabled=True; IlfCommand=SLIN
;ENDFOLD
SLIN XP369 WITH $VEL = SVEL_CP(2.0, , LCPDAT369),$TOOL = STOOL2(FP369),$BASE = SBASE(FP369.BASE_NO),$IPO_MODE = SIPO_MODE(FP369.IPO_FRAME),$LOAD = SLOAD(FP369.TOOL_NO),$ACC = SACC_CP(LCPDAT369),$ORI_TYPE = SORI_TYP(LCPDAT369),$APO = SAPO(LCPDAT369),$JERK = SJERK(LCPDAT369),$COLLMON_TOL_PRO[1] = USE_CM_PRO_VALUES(0)
;ENDFOLD

;FOLD SLIN P370 Vel=1 m/s CPDAT370 Tool[4]:Microflown3D Base[0];%{PE}
;FOLD Parameters ;%{h}
;Params IlfProvider=kukaroboter.basistech.inlineforms.movement.spline; Kuka.IsGlobalPoint=False; Kuka.PointName=P370; Kuka.BlendingEnabled=False; Kuka.MoveDataName=CPDAT370; Kuka.VelocityPath=1.000; Kuka.VelocityFieldEnabled=True; Kuka.ColDetectFieldEnabled=True; Kuka.CurrentCDSetIndex=0; Kuka.MovementParameterFieldEnabled=True; IlfCommand=SLIN
;ENDFOLD
SLIN XP370 WITH $VEL = SVEL_CP(2.0, , LCPDAT370),$TOOL = STOOL2(FP370),$BASE = SBASE(FP370.BASE_NO),$IPO_MODE = SIPO_MODE(FP370.IPO_FRAME),$LOAD = SLOAD(FP370.TOOL_NO),$ACC = SACC_CP(LCPDAT370),$ORI_TYPE = SORI_TYP(LCPDAT370),$APO = SAPO(LCPDAT370),$JERK = SJERK(LCPDAT370),$COLLMON_TOL_PRO[1] = USE_CM_PRO_VALUES(0)
;ENDFOLD

;FOLD SLIN P371 Vel=1 m/s CPDAT371 Tool[4]:Microflown3D Base[0];%{PE}
;FOLD Parameters ;%{h}
;Params IlfProvider=kukaroboter.basistech.inlineforms.movement.spline; Kuka.IsGlobalPoint=False; Kuka.PointName=P371; Kuka.BlendingEnabled=False; Kuka.MoveDataName=CPDAT371; Kuka.VelocityPath=1.000; Kuka.VelocityFieldEnabled=True; Kuka.ColDetectFieldEnabled=True; Kuka.CurrentCDSetIndex=0; Kuka.MovementParameterFieldEnabled=True; IlfCommand=SLIN
;ENDFOLD
SLIN XP371 WITH $VEL = SVEL_CP(2.0, , LCPDAT371),$TOOL = STOOL2(FP371),$BASE = SBASE(FP371.BASE_NO),$IPO_MODE = SIPO_MODE(FP371.IPO_FRAME),$LOAD = SLOAD(FP371.TOOL_NO),$ACC = SACC_CP(LCPDAT371),$ORI_TYPE = SORI_TYP(LCPDAT371),$APO = SAPO(LCPDAT371),$JERK = SJERK(LCPDAT371),$COLLMON_TOL_PRO[1] = USE_CM_PRO_VALUES(0)
;ENDFOLD

;FOLD SLIN P372 Vel=1 m/s CPDAT372 Tool[4]:Microflown3D Base[0];%{PE}
;FOLD Parameters ;%{h}
;Params IlfProvider=kukaroboter.basistech.inlineforms.movement.spline; Kuka.IsGlobalPoint=False; Kuka.PointName=P372; Kuka.BlendingEnabled=False; Kuka.MoveDataName=CPDAT372; Kuka.VelocityPath=1.000; Kuka.VelocityFieldEnabled=True; Kuka.ColDetectFieldEnabled=True; Kuka.CurrentCDSetIndex=0; Kuka.MovementParameterFieldEnabled=True; IlfCommand=SLIN
;ENDFOLD
SLIN XP372 WITH $VEL = SVEL_CP(2.0, , LCPDAT372),$TOOL = STOOL2(FP372),$BASE = SBASE(FP372.BASE_NO),$IPO_MODE = SIPO_MODE(FP372.IPO_FRAME),$LOAD = SLOAD(FP372.TOOL_NO),$ACC = SACC_CP(LCPDAT372),$ORI_TYPE = SORI_TYP(LCPDAT372),$APO = SAPO(LCPDAT372),$JERK = SJERK(LCPDAT372),$COLLMON_TOL_PRO[1] = USE_CM_PRO_VALUES(0)
;ENDFOLD

;FOLD SLIN P373 Vel=1 m/s CPDAT373 Tool[4]:Microflown3D Base[0];%{PE}
;FOLD Parameters ;%{h}
;Params IlfProvider=kukaroboter.basistech.inlineforms.movement.spline; Kuka.IsGlobalPoint=False; Kuka.PointName=P373; Kuka.BlendingEnabled=False; Kuka.MoveDataName=CPDAT373; Kuka.VelocityPath=1.000; Kuka.VelocityFieldEnabled=True; Kuka.ColDetectFieldEnabled=True; Kuka.CurrentCDSetIndex=0; Kuka.MovementParameterFieldEnabled=True; IlfCommand=SLIN
;ENDFOLD
SLIN XP373 WITH $VEL = SVEL_CP(2.0, , LCPDAT373),$TOOL = STOOL2(FP373),$BASE = SBASE(FP373.BASE_NO),$IPO_MODE = SIPO_MODE(FP373.IPO_FRAME),$LOAD = SLOAD(FP373.TOOL_NO),$ACC = SACC_CP(LCPDAT373),$ORI_TYPE = SORI_TYP(LCPDAT373),$APO = SAPO(LCPDAT373),$JERK = SJERK(LCPDAT373),$COLLMON_TOL_PRO[1] = USE_CM_PRO_VALUES(0)
;ENDFOLD

;FOLD SLIN P374 Vel=1 m/s CPDAT374 Tool[4]:Microflown3D Base[0];%{PE}
;FOLD Parameters ;%{h}
;Params IlfProvider=kukaroboter.basistech.inlineforms.movement.spline; Kuka.IsGlobalPoint=False; Kuka.PointName=P374; Kuka.BlendingEnabled=False; Kuka.MoveDataName=CPDAT374; Kuka.VelocityPath=1.000; Kuka.VelocityFieldEnabled=True; Kuka.ColDetectFieldEnabled=True; Kuka.CurrentCDSetIndex=0; Kuka.MovementParameterFieldEnabled=True; IlfCommand=SLIN
;ENDFOLD
SLIN XP374 WITH $VEL = SVEL_CP(2.0, , LCPDAT374),$TOOL = STOOL2(FP374),$BASE = SBASE(FP374.BASE_NO),$IPO_MODE = SIPO_MODE(FP374.IPO_FRAME),$LOAD = SLOAD(FP374.TOOL_NO),$ACC = SACC_CP(LCPDAT374),$ORI_TYPE = SORI_TYP(LCPDAT374),$APO = SAPO(LCPDAT374),$JERK = SJERK(LCPDAT374),$COLLMON_TOL_PRO[1] = USE_CM_PRO_VALUES(0)
;ENDFOLD

;FOLD SLIN P375 Vel=1 m/s CPDAT375 Tool[4]:Microflown3D Base[0];%{PE}
;FOLD Parameters ;%{h}
;Params IlfProvider=kukaroboter.basistech.inlineforms.movement.spline; Kuka.IsGlobalPoint=False; Kuka.PointName=P375; Kuka.BlendingEnabled=False; Kuka.MoveDataName=CPDAT375; Kuka.VelocityPath=1.000; Kuka.VelocityFieldEnabled=True; Kuka.ColDetectFieldEnabled=True; Kuka.CurrentCDSetIndex=0; Kuka.MovementParameterFieldEnabled=True; IlfCommand=SLIN
;ENDFOLD
SLIN XP375 WITH $VEL = SVEL_CP(2.0, , LCPDAT375),$TOOL = STOOL2(FP375),$BASE = SBASE(FP375.BASE_NO),$IPO_MODE = SIPO_MODE(FP375.IPO_FRAME),$LOAD = SLOAD(FP375.TOOL_NO),$ACC = SACC_CP(LCPDAT375),$ORI_TYPE = SORI_TYP(LCPDAT375),$APO = SAPO(LCPDAT375),$JERK = SJERK(LCPDAT375),$COLLMON_TOL_PRO[1] = USE_CM_PRO_VALUES(0)
;ENDFOLD

;FOLD SLIN P376 Vel=1 m/s CPDAT376 Tool[4]:Microflown3D Base[0];%{PE}
;FOLD Parameters ;%{h}
;Params IlfProvider=kukaroboter.basistech.inlineforms.movement.spline; Kuka.IsGlobalPoint=False; Kuka.PointName=P376; Kuka.BlendingEnabled=False; Kuka.MoveDataName=CPDAT376; Kuka.VelocityPath=1.000; Kuka.VelocityFieldEnabled=True; Kuka.ColDetectFieldEnabled=True; Kuka.CurrentCDSetIndex=0; Kuka.MovementParameterFieldEnabled=True; IlfCommand=SLIN
;ENDFOLD
SLIN XP376 WITH $VEL = SVEL_CP(2.0, , LCPDAT376),$TOOL = STOOL2(FP376),$BASE = SBASE(FP376.BASE_NO),$IPO_MODE = SIPO_MODE(FP376.IPO_FRAME),$LOAD = SLOAD(FP376.TOOL_NO),$ACC = SACC_CP(LCPDAT376),$ORI_TYPE = SORI_TYP(LCPDAT376),$APO = SAPO(LCPDAT376),$JERK = SJERK(LCPDAT376),$COLLMON_TOL_PRO[1] = USE_CM_PRO_VALUES(0)
;ENDFOLD

;FOLD SLIN P377 Vel=1 m/s CPDAT377 Tool[4]:Microflown3D Base[0];%{PE}
;FOLD Parameters ;%{h}
;Params IlfProvider=kukaroboter.basistech.inlineforms.movement.spline; Kuka.IsGlobalPoint=False; Kuka.PointName=P377; Kuka.BlendingEnabled=False; Kuka.MoveDataName=CPDAT377; Kuka.VelocityPath=1.000; Kuka.VelocityFieldEnabled=True; Kuka.ColDetectFieldEnabled=True; Kuka.CurrentCDSetIndex=0; Kuka.MovementParameterFieldEnabled=True; IlfCommand=SLIN
;ENDFOLD
SLIN XP377 WITH $VEL = SVEL_CP(2.0, , LCPDAT377),$TOOL = STOOL2(FP377),$BASE = SBASE(FP377.BASE_NO),$IPO_MODE = SIPO_MODE(FP377.IPO_FRAME),$LOAD = SLOAD(FP377.TOOL_NO),$ACC = SACC_CP(LCPDAT377),$ORI_TYPE = SORI_TYP(LCPDAT377),$APO = SAPO(LCPDAT377),$JERK = SJERK(LCPDAT377),$COLLMON_TOL_PRO[1] = USE_CM_PRO_VALUES(0)
;ENDFOLD

;FOLD SLIN P378 Vel=1 m/s CPDAT378 Tool[4]:Microflown3D Base[0];%{PE}
;FOLD Parameters ;%{h}
;Params IlfProvider=kukaroboter.basistech.inlineforms.movement.spline; Kuka.IsGlobalPoint=False; Kuka.PointName=P378; Kuka.BlendingEnabled=False; Kuka.MoveDataName=CPDAT378; Kuka.VelocityPath=1.000; Kuka.VelocityFieldEnabled=True; Kuka.ColDetectFieldEnabled=True; Kuka.CurrentCDSetIndex=0; Kuka.MovementParameterFieldEnabled=True; IlfCommand=SLIN
;ENDFOLD
SLIN XP378 WITH $VEL = SVEL_CP(2.0, , LCPDAT378),$TOOL = STOOL2(FP378),$BASE = SBASE(FP378.BASE_NO),$IPO_MODE = SIPO_MODE(FP378.IPO_FRAME),$LOAD = SLOAD(FP378.TOOL_NO),$ACC = SACC_CP(LCPDAT378),$ORI_TYPE = SORI_TYP(LCPDAT378),$APO = SAPO(LCPDAT378),$JERK = SJERK(LCPDAT378),$COLLMON_TOL_PRO[1] = USE_CM_PRO_VALUES(0)
;ENDFOLD

;FOLD SLIN P379 Vel=1 m/s CPDAT379 Tool[4]:Microflown3D Base[0];%{PE}
;FOLD Parameters ;%{h}
;Params IlfProvider=kukaroboter.basistech.inlineforms.movement.spline; Kuka.IsGlobalPoint=False; Kuka.PointName=P379; Kuka.BlendingEnabled=False; Kuka.MoveDataName=CPDAT379; Kuka.VelocityPath=1.000; Kuka.VelocityFieldEnabled=True; Kuka.ColDetectFieldEnabled=True; Kuka.CurrentCDSetIndex=0; Kuka.MovementParameterFieldEnabled=True; IlfCommand=SLIN
;ENDFOLD
SLIN XP379 WITH $VEL = SVEL_CP(2.0, , LCPDAT379),$TOOL = STOOL2(FP379),$BASE = SBASE(FP379.BASE_NO),$IPO_MODE = SIPO_MODE(FP379.IPO_FRAME),$LOAD = SLOAD(FP379.TOOL_NO),$ACC = SACC_CP(LCPDAT379),$ORI_TYPE = SORI_TYP(LCPDAT379),$APO = SAPO(LCPDAT379),$JERK = SJERK(LCPDAT379),$COLLMON_TOL_PRO[1] = USE_CM_PRO_VALUES(0)
;ENDFOLD

;FOLD SLIN P380 Vel=1 m/s CPDAT380 Tool[4]:Microflown3D Base[0];%{PE}
;FOLD Parameters ;%{h}
;Params IlfProvider=kukaroboter.basistech.inlineforms.movement.spline; Kuka.IsGlobalPoint=False; Kuka.PointName=P380; Kuka.BlendingEnabled=False; Kuka.MoveDataName=CPDAT380; Kuka.VelocityPath=1.000; Kuka.VelocityFieldEnabled=True; Kuka.ColDetectFieldEnabled=True; Kuka.CurrentCDSetIndex=0; Kuka.MovementParameterFieldEnabled=True; IlfCommand=SLIN
;ENDFOLD
SLIN XP380 WITH $VEL = SVEL_CP(2.0, , LCPDAT380),$TOOL = STOOL2(FP380),$BASE = SBASE(FP380.BASE_NO),$IPO_MODE = SIPO_MODE(FP380.IPO_FRAME),$LOAD = SLOAD(FP380.TOOL_NO),$ACC = SACC_CP(LCPDAT380),$ORI_TYPE = SORI_TYP(LCPDAT380),$APO = SAPO(LCPDAT380),$JERK = SJERK(LCPDAT380),$COLLMON_TOL_PRO[1] = USE_CM_PRO_VALUES(0)
;ENDFOLD

;FOLD SLIN P381 Vel=1 m/s CPDAT381 Tool[4]:Microflown3D Base[0];%{PE}
;FOLD Parameters ;%{h}
;Params IlfProvider=kukaroboter.basistech.inlineforms.movement.spline; Kuka.IsGlobalPoint=False; Kuka.PointName=P381; Kuka.BlendingEnabled=False; Kuka.MoveDataName=CPDAT381; Kuka.VelocityPath=1.000; Kuka.VelocityFieldEnabled=True; Kuka.ColDetectFieldEnabled=True; Kuka.CurrentCDSetIndex=0; Kuka.MovementParameterFieldEnabled=True; IlfCommand=SLIN
;ENDFOLD
SLIN XP381 WITH $VEL = SVEL_CP(2.0, , LCPDAT381),$TOOL = STOOL2(FP381),$BASE = SBASE(FP381.BASE_NO),$IPO_MODE = SIPO_MODE(FP381.IPO_FRAME),$LOAD = SLOAD(FP381.TOOL_NO),$ACC = SACC_CP(LCPDAT381),$ORI_TYPE = SORI_TYP(LCPDAT381),$APO = SAPO(LCPDAT381),$JERK = SJERK(LCPDAT381),$COLLMON_TOL_PRO[1] = USE_CM_PRO_VALUES(0)
;ENDFOLD

;FOLD SLIN P382 Vel=1 m/s CPDAT382 Tool[4]:Microflown3D Base[0];%{PE}
;FOLD Parameters ;%{h}
;Params IlfProvider=kukaroboter.basistech.inlineforms.movement.spline; Kuka.IsGlobalPoint=False; Kuka.PointName=P382; Kuka.BlendingEnabled=False; Kuka.MoveDataName=CPDAT382; Kuka.VelocityPath=1.000; Kuka.VelocityFieldEnabled=True; Kuka.ColDetectFieldEnabled=True; Kuka.CurrentCDSetIndex=0; Kuka.MovementParameterFieldEnabled=True; IlfCommand=SLIN
;ENDFOLD
SLIN XP382 WITH $VEL = SVEL_CP(2.0, , LCPDAT382),$TOOL = STOOL2(FP382),$BASE = SBASE(FP382.BASE_NO),$IPO_MODE = SIPO_MODE(FP382.IPO_FRAME),$LOAD = SLOAD(FP382.TOOL_NO),$ACC = SACC_CP(LCPDAT382),$ORI_TYPE = SORI_TYP(LCPDAT382),$APO = SAPO(LCPDAT382),$JERK = SJERK(LCPDAT382),$COLLMON_TOL_PRO[1] = USE_CM_PRO_VALUES(0)
;ENDFOLD

;FOLD SLIN P383 Vel=1 m/s CPDAT383 Tool[4]:Microflown3D Base[0];%{PE}
;FOLD Parameters ;%{h}
;Params IlfProvider=kukaroboter.basistech.inlineforms.movement.spline; Kuka.IsGlobalPoint=False; Kuka.PointName=P383; Kuka.BlendingEnabled=False; Kuka.MoveDataName=CPDAT383; Kuka.VelocityPath=1.000; Kuka.VelocityFieldEnabled=True; Kuka.ColDetectFieldEnabled=True; Kuka.CurrentCDSetIndex=0; Kuka.MovementParameterFieldEnabled=True; IlfCommand=SLIN
;ENDFOLD
SLIN XP383 WITH $VEL = SVEL_CP(2.0, , LCPDAT383),$TOOL = STOOL2(FP383),$BASE = SBASE(FP383.BASE_NO),$IPO_MODE = SIPO_MODE(FP383.IPO_FRAME),$LOAD = SLOAD(FP383.TOOL_NO),$ACC = SACC_CP(LCPDAT383),$ORI_TYPE = SORI_TYP(LCPDAT383),$APO = SAPO(LCPDAT383),$JERK = SJERK(LCPDAT383),$COLLMON_TOL_PRO[1] = USE_CM_PRO_VALUES(0)
;ENDFOLD

;FOLD SLIN P384 Vel=1 m/s CPDAT384 Tool[4]:Microflown3D Base[0];%{PE}
;FOLD Parameters ;%{h}
;Params IlfProvider=kukaroboter.basistech.inlineforms.movement.spline; Kuka.IsGlobalPoint=False; Kuka.PointName=P384; Kuka.BlendingEnabled=False; Kuka.MoveDataName=CPDAT384; Kuka.VelocityPath=1.000; Kuka.VelocityFieldEnabled=True; Kuka.ColDetectFieldEnabled=True; Kuka.CurrentCDSetIndex=0; Kuka.MovementParameterFieldEnabled=True; IlfCommand=SLIN
;ENDFOLD
SLIN XP384 WITH $VEL = SVEL_CP(2.0, , LCPDAT384),$TOOL = STOOL2(FP384),$BASE = SBASE(FP384.BASE_NO),$IPO_MODE = SIPO_MODE(FP384.IPO_FRAME),$LOAD = SLOAD(FP384.TOOL_NO),$ACC = SACC_CP(LCPDAT384),$ORI_TYPE = SORI_TYP(LCPDAT384),$APO = SAPO(LCPDAT384),$JERK = SJERK(LCPDAT384),$COLLMON_TOL_PRO[1] = USE_CM_PRO_VALUES(0)
;ENDFOLD

